C07304=1167.739,85.707,-51.427,-179.195,6.255,148.894
C07305=1167.744,85.458,-51.409,-179.197,6.253,148.894
C07306=1167.749,85.208,-51.392,-179.200,6.251,148.895
C07307=1167.754,84.959,-51.374,-179.203,6.251,148.895
C07308=1167.760,84.709,-51.357,-179.205,6.249,148.896
C07309=1167.764,84.460,-51.339,-179.208,6.248,148.896
C07310=1167.769,84.211,-51.321,-179.211,6.247,148.897
C07311=1167.774,83.961,-51.304,-179.213,6.246,148.897
C07312=1167.779,83.712,-51.286,-179.216,6.245,148.898
C07313=1167.784,83.463,-51.270,-179.218,6.244,148.898
C07314=1167.789,83.214,-51.252,-179.221,6.242,148.899
C07315=1167.794,82.964,-51.235,-179.224,6.241,148.899
C07316=1167.798,82.716,-51.217,-179.226,6.240,148.900
C07317=1167.803,82.466,-51.200,-179.230,6.239,148.900
C07318=1167.808,82.217,-51.182,-179.232,6.238,148.901
C07319=1167.813,81.967,-51.165,-179.234,6.236,148.901
C07320=1167.818,81.718,-51.147,-179.237,6.236,148.902
C07321=1167.823,81.468,-51.130,-179.240,6.234,148.902
C07322=1167.828,81.218,-51.113,-179.242,6.233,148.903
C07323=1167.832,80.969,-51.096,-179.245,6.232,148.903
C07324=1167.838,80.720,-51.079,-179.248,6.230,148.904
C07325=1167.843,80.452,-51.060,-179.250,6.229,148.904
C07326=1167.848,80.184,-51.041,-179.254,6.228,148.905
C07327=1167.854,79.915,-51.023,-179.256,6.226,148.905
C07328=1167.859,79.647,-51.004,-179.259,6.226,148.906
C07329=1167.863,79.398,-50.987,-179.262,6.224,148.907
C07330=1167.869,79.148,-50.969,-179.264,6.224,148.907
C07331=1167.874,78.898,-50.952,-179.267,6.222,148.908
C07332=1167.878,78.649,-50.935,-179.270,6.220,148.908
C07333=1167.884,78.400,-50.918,-179.272,6.220,148.909
C07334=1167.888,78.151,-50.901,-179.275,6.218,148.909
C07335=1167.893,77.901,-50.883,-179.278,6.218,148.910
C07336=1167.898,77.652,-50.866,-179.281,6.216,148.910
C07337=1167.903,77.402,-50.849,-179.283,6.215,148.911
C07338=1167.909,77.153,-50.832,-179.286,6.214,148.911
C07339=1167.913,76.904,-50.815,-179.288,6.213,148.912
C07340=1167.918,76.654,-50.798,-179.291,6.211,148.912
C07341=1167.923,76.405,-50.781,-179.293,6.211,148.913
C07342=1167.928,76.155,-50.764,-179.297,6.209,148.913
C07343=1167.932,75.906,-50.746,-179.299,6.208,148.914
C07344=1167.938,75.657,-50.730,-179.302,6.207,148.914
C07345=1167.942,75.408,-50.713,-179.304,6.206,148.915
C07346=1167.947,75.158,-50.696,-179.307,6.204,148.915
C07347=1167.952,74.908,-50.679,-179.310,6.204,148.916
C07348=1167.957,74.660,-50.661,-179.312,6.202,148.917
C07349=1167.962,74.410,-50.645,-179.315,6.202,148.917
C07350=1167.967,74.161,-50.627,-179.318,6.200,148.918
C07351=1167.972,73.911,-50.611,-179.320,6.199,148.918
C07352=1167.977,73.662,-50.594,-179.323,6.198,148.919
C07353=1167.982,73.413,-50.577,-179.325,6.197,148.919
C07354=1167.987,73.163,-50.560,-179.328,6.196,148.920
C07355=1167.991,72.914,-50.542,-179.330,6.195,148.920
C07356=1167.997,72.665,-50.526,-179.334,6.193,148.921
C07357=1168.002,72.415,-50.509,-179.336,6.192,148.921
C07358=1168.007,72.166,-50.492,-179.339,6.191,148.922
C07359=1168.011,71.916,-50.475,-179.341,6.190,148.922
C07360=1168.016,71.667,-50.459,-179.344,6.189,148.923
C07361=1168.022,71.418,-50.441,-179.347,6.188,148.923
C07362=1168.026,71.168,-50.425,-179.349,6.186,148.924
C07363=1168.031,70.918,-50.407,-179.352,6.186,148.925
C07364=1168.036,70.669,-50.391,-179.354,6.185,148.925
C07365=1168.041,70.420,-50.375,-179.357,6.184,148.926
C07366=1168.046,70.170,-50.357,-179.359,6.183,148.926
C07367=1168.051,69.921,-50.341,-179.362,6.181,148.927
C07368=1168.056,69.672,-50.324,-179.365,6.181,148.927
C07369=1168.061,69.422,-50.307,-179.368,6.179,148.928
C07370=1168.066,69.173,-50.291,-179.370,6.178,148.928
C07371=1168.071,68.924,-50.273,-179.373,6.177,148.929
C07372=1168.076,68.674,-50.257,-179.376,6.176,148.929
C07373=1168.081,68.425,-50.240,-179.378,6.175,148.930
C07374=1168.085,68.176,-50.224,-179.381,6.174,148.930
C07375=1168.090,67.926,-50.207,-179.384,6.172,148.931
C07376=1168.096,67.677,-50.190,-179.386,6.172,148.932
C07377=1168.100,67.427,-50.174,-179.388,6.171,148.932
C07378=1168.106,67.177,-50.157,-179.391,6.169,148.932
C07379=1168.111,66.929,-50.141,-179.394,6.169,148.933
C07380=1168.115,66.679,-50.124,-179.397,6.167,148.933
C07381=1168.120,66.429,-50.107,-179.399,6.167,148.934
C07382=1168.125,66.180,-50.090,-179.402,6.165,148.935
C07383=1168.130,65.931,-50.074,-179.405,6.164,148.935
C07384=1168.135,65.682,-50.058,-179.407,6.163,148.936
C07385=1168.140,65.432,-50.041,-179.410,6.162,148.936
C07386=1168.145,65.182,-50.024,-179.412,6.161,148.937
C07387=1168.150,64.934,-50.008,-179.415,6.160,148.937
C07388=1168.155,64.684,-49.991,-179.417,6.159,148.938
C07389=1168.160,64.435,-49.976,-179.421,6.158,148.939
C07390=1168.165,64.185,-49.958,-179.423,6.157,148.939
C07391=1168.170,63.935,-49.942,-179.426,6.156,148.940
C07392=1168.175,63.687,-49.926,-179.428,6.155,148.940
C07393=1168.179,63.436,-49.910,-179.431,6.153,148.940
C07394=1168.185,63.188,-49.893,-179.434,6.152,148.941
C07395=1168.190,62.938,-49.876,-179.436,6.152,148.942
C07396=1168.194,62.688,-49.859,-179.439,6.150,148.942
C07397=1168.200,62.439,-49.844,-179.441,6.149,148.943
C07398=1168.204,62.190,-49.827,-179.444,6.148,148.943
C07399=1168.209,61.941,-49.811,-179.446,6.147,148.944
C07400=1168.214,61.691,-49.795,-179.449,6.147,148.944
C07401=1168.220,61.442,-49.778,-179.452,6.145,148.945
C07402=1168.224,61.192,-49.761,-179.454,6.145,148.946
C07403=1168.230,60.943,-49.746,-179.457,6.143,148.946
C07404=1168.234,60.693,-49.729,-179.460,6.142,148.947
C07405=1168.239,60.444,-49.713,-179.462,6.141,148.947
C07406=1168.244,60.194,-49.697,-179.465,6.140,148.948
C07407=1168.249,59.946,-49.680,-179.467,6.139,148.948
C07408=1168.254,59.695,-49.664,-179.471,6.138,148.949
C07409=1168.259,59.447,-49.648,-179.473,6.137,148.949
C07410=1168.264,59.197,-49.631,-179.476,6.136,148.950
C07411=1168.270,58.947,-49.615,-179.478,6.135,148.950
C07412=1168.274,58.698,-49.599,-179.481,6.134,148.951
C07413=1168.279,58.449,-49.583,-179.483,6.133,148.951
C07414=1168.284,58.199,-49.566,-179.486,6.132,148.952
C07415=1168.289,57.950,-49.551,-179.488,6.131,148.953
C07416=1168.294,57.700,-49.534,-179.491,6.130,148.953
C07417=1168.299,57.451,-49.519,-179.494,6.129,148.954
C07418=1168.304,57.201,-49.502,-179.497,6.128,148.954
C07419=1168.309,56.952,-49.486,-179.499,6.127,148.955
C07420=1168.314,56.702,-49.470,-179.502,6.127,148.955
C07421=1168.319,56.453,-49.454,-179.504,6.125,148.956
C07422=1168.323,56.204,-49.437,-179.507,6.124,148.957
C07423=1168.329,55.954,-49.422,-179.510,6.123,148.957
C07424=1168.333,55.705,-49.405,-179.512,6.122,148.958
C07425=1168.339,55.455,-49.390,-179.515,6.121,148.958
C07426=1168.344,55.206,-49.373,-179.518,6.120,148.959
C07427=1168.349,54.956,-49.357,-179.520,6.119,148.959
C07428=1168.354,54.707,-49.342,-179.523,6.119,148.960
C07429=1168.359,54.438,-49.324,-179.525,6.117,148.960
C07430=1168.364,54.170,-49.307,-179.529,6.116,148.961
C07431=1168.370,53.901,-49.290,-179.531,6.115,148.962
C07432=1168.375,53.633,-49.273,-179.534,6.113,148.962
C07433=1168.380,53.383,-49.257,-179.537,6.113,148.963
C07434=1168.385,53.134,-49.240,-179.539,6.112,148.963
C07435=1168.390,52.885,-49.225,-179.542,6.111,148.964
C07436=1168.395,52.635,-49.209,-179.544,6.110,148.964
C07437=1168.400,52.386,-49.192,-179.547,6.109,148.965
C07438=1168.405,52.136,-49.176,-179.549,6.108,148.965
C07439=1168.410,51.887,-49.161,-179.552,6.107,148.966
C07440=1168.415,51.638,-49.145,-179.554,6.106,148.967
C07441=1168.420,51.388,-49.129,-179.557,6.105,148.967
C07442=1168.425,51.138,-49.114,-179.560,6.104,148.968
C07443=1168.430,50.889,-49.097,-179.562,6.104,148.968
C07444=1168.435,50.639,-49.081,-179.565,6.102,148.969
C07445=1168.440,50.390,-49.066,-179.568,6.102,148.969
C07446=1168.444,50.140,-49.050,-179.570,6.100,148.970
C07447=1168.449,49.891,-49.034,-179.573,6.099,148.971
C07448=1168.455,49.642,-49.019,-179.576,6.099,148.971
C07449=1168.460,49.392,-49.003,-179.578,6.097,148.972
C07450=1168.465,49.142,-48.987,-179.581,6.097,148.972
C07451=1168.470,48.893,-48.971,-179.583,6.096,148.973
C07452=1168.474,48.644,-48.955,-179.586,6.095,148.973
C07453=1168.479,48.395,-48.940,-179.589,6.094,148.974
C07454=1168.485,48.145,-48.924,-179.591,6.093,148.975
C07455=1168.490,47.895,-48.908,-179.594,6.091,148.975
C07456=1168.495,47.646,-48.893,-179.597,6.091,148.976
C07457=1168.500,47.397,-48.878,-179.599,6.090,148.976
C07458=1168.505,47.147,-48.862,-179.601,6.090,148.977
C07459=1168.510,46.898,-48.845,-179.604,6.088,148.977
C07460=1168.515,46.648,-48.830,-179.607,6.087,148.978
C07461=1168.520,46.399,-48.815,-179.609,6.087,148.978
C07462=1168.524,46.149,-48.799,-179.612,6.085,148.979
C07463=1168.530,45.900,-48.783,-179.614,6.084,148.979
C07464=1168.535,45.650,-48.768,-179.617,6.084,148.980
C07465=1168.540,45.401,-48.753,-179.620,6.082,148.981
C07466=1168.545,45.151,-48.737,-179.622,6.082,148.981
C07467=1168.550,44.902,-48.721,-179.624,6.081,148.982
C07468=1168.555,44.653,-48.706,-179.628,6.080,148.982
C07469=1168.559,44.402,-48.690,-179.630,6.079,148.983
C07470=1168.565,44.153,-48.675,-179.633,6.078,148.983
C07471=1168.570,43.904,-48.659,-179.636,6.077,148.984
C07472=1168.575,43.655,-48.644,-179.638,6.076,148.985
C07473=1168.580,43.405,-48.628,-179.641,6.076,148.985
C07474=1168.585,43.155,-48.612,-179.643,6.075,148.986
C07475=1168.590,42.906,-48.597,-179.646,6.073,148.986
C07476=1168.595,42.657,-48.582,-179.648,6.073,148.987
C07477=1168.600,42.407,-48.566,-179.651,6.072,148.987
C07478=1168.604,42.157,-48.551,-179.653,6.070,148.988
C07479=1168.610,41.908,-48.535,-179.656,6.070,148.989
C07480=1168.615,41.659,-48.520,-179.658,6.069,148.989
C07481=1168.620,41.409,-48.505,-179.661,6.069,148.990
C07482=1168.625,41.160,-48.489,-179.664,6.067,148.990
C07483=1168.629,40.910,-48.474,-179.666,6.066,148.991
C07484=1168.635,40.661,-48.458,-179.669,6.066,148.991
C07485=1168.640,40.411,-48.443,-179.672,6.064,148.992
C07486=1168.645,40.162,-48.428,-179.674,6.064,148.993
C07487=1168.650,39.912,-48.413,-179.676,6.063,148.993
C07488=1168.655,39.663,-48.398,-179.679,6.062,148.994
C07489=1168.660,39.413,-48.382,-179.682,6.061,148.994
C07490=1168.665,39.164,-48.367,-179.685,6.060,148.995
C07491=1168.670,38.915,-48.351,-179.687,6.059,148.995
C07492=1168.675,38.665,-48.336,-179.690,6.058,148.996
C07493=1168.680,38.416,-48.321,-179.693,6.058,148.997
C07494=1168.686,38.166,-48.306,-179.695,6.057,148.997
C07495=1168.690,37.916,-48.290,-179.697,6.056,148.998
C07496=1168.695,37.667,-48.275,-179.700,6.055,148.998
C07497=1168.700,37.417,-48.261,-179.703,6.054,148.999
C07498=1168.705,37.168,-48.245,-179.705,6.053,148.999
C07499=1168.710,36.919,-48.230,-179.708,6.053,149.000
C07500=1168.715,36.669,-48.214,-179.710,6.051,149.000
C07501=1168.720,36.420,-48.200,-179.713,6.051,149.001
C07502=1168.726,36.170,-48.185,-179.716,6.050,149.002
C07503=1168.730,35.920,-48.169,-179.718,6.049,149.002
C07504=1168.735,35.671,-48.154,-179.721,6.048,149.003
C07505=1168.740,35.421,-48.139,-179.723,6.047,149.003
C07506=1168.746,35.172,-48.124,-179.726,6.047,149.004
C07507=1168.750,34.923,-48.109,-179.728,6.046,149.004
C07508=1168.756,34.673,-48.094,-179.731,6.045,149.005
C07509=1168.761,34.424,-48.079,-179.733,6.044,149.006
C07510=1168.766,34.174,-48.063,-179.736,6.043,149.006
C07511=1168.771,33.925,-48.049,-179.739,6.043,149.007
C07512=1168.776,33.676,-48.034,-179.741,6.041,149.007
C07513=1168.781,33.426,-48.018,-179.744,6.041,149.008
C07514=1168.786,33.176,-48.004,-179.746,6.040,149.009
C07515=1168.791,32.927,-47.989,-179.749,6.039,149.009
C07516=1168.795,32.677,-47.973,-179.752,6.038,149.010
C07517=1168.800,32.427,-47.959,-179.754,6.037,149.010
C07518=1168.806,32.178,-47.943,-179.756,6.036,149.011
C07519=1168.811,31.928,-47.929,-179.759,6.036,149.011
C07520=1168.816,31.679,-47.913,-179.762,6.035,149.012
C07521=1168.821,31.429,-47.899,-179.764,6.034,149.013
C07522=1168.826,31.180,-47.884,-179.767,6.033,149.013
C07523=1168.831,30.931,-47.869,-179.769,6.032,149.014
C07524=1168.836,30.681,-47.854,-179.772,6.032,149.014
C07525=1168.841,30.432,-47.839,-179.775,6.030,149.015
C07526=1168.846,30.182,-47.824,-179.777,6.030,149.016
C07527=1168.851,29.933,-47.809,-179.780,6.029,149.016
C07528=1168.856,29.683,-47.795,-179.782,6.028,149.017
C07529=1168.861,29.434,-47.780,-179.785,6.028,149.017
C07530=1168.866,29.184,-47.765,-179.787,6.026,149.018
C07531=1168.871,28.935,-47.750,-179.790,6.026,149.018
C07532=1168.877,28.685,-47.735,-179.792,6.025,149.019
C07533=1168.882,28.416,-47.720,-179.795,6.024,149.020
C07534=1168.887,28.147,-47.704,-179.798,6.023,149.020
C07535=1168.893,27.878,-47.688,-179.801,6.023,149.021
C07536=1168.898,27.609,-47.672,-179.804,6.021,149.021
C07537=1168.903,27.360,-47.658,-179.806,6.020,149.022
C07538=1168.908,27.110,-47.642,-179.809,6.020,149.023
C07539=1168.913,26.861,-47.628,-179.811,6.019,149.023
C07540=1168.918,26.612,-47.613,-179.814,6.019,149.024
C07541=1168.923,26.363,-47.599,-179.816,6.017,149.024
C07542=1168.929,26.112,-47.584,-179.819,6.016,149.025
C07543=1168.934,25.863,-47.569,-179.822,6.016,149.026
C07544=1168.939,25.614,-47.555,-179.824,6.015,149.026
C07545=1168.944,25.364,-47.541,-179.827,6.015,149.027
C07546=1168.949,25.115,-47.525,-179.829,6.013,149.027
C07547=1168.954,24.865,-47.511,-179.832,6.013,149.028
C07548=1168.959,24.615,-47.496,-179.834,6.012,149.028
C07549=1168.964,24.366,-47.481,-179.837,6.011,149.029
C07550=1168.968,24.116,-47.467,-179.839,6.011,149.030
C07551=1168.974,23.866,-47.452,-179.842,6.010,149.030
C07552=1168.979,23.617,-47.437,-179.845,6.009,149.031
C07553=1168.984,23.368,-47.423,-179.847,6.008,149.031
C07554=1168.989,23.119,-47.409,-179.850,6.007,149.032
C07555=1168.994,22.869,-47.395,-179.852,6.006,149.032
C07556=1168.999,22.620,-47.380,-179.854,6.006,149.033
C07557=1169.005,22.370,-47.365,-179.857,6.005,149.034
C07558=1169.010,22.120,-47.351,-179.860,6.004,149.034
C07559=1169.015,21.870,-47.336,-179.862,6.003,149.035
C07560=1169.019,21.621,-47.321,-179.865,6.003,149.035
C07561=1169.024,21.371,-47.307,-179.867,6.002,149.036
C07562=1169.029,21.122,-47.293,-179.870,6.002,149.037
C07563=1169.035,20.873,-47.279,-179.872,6.001,149.037
C07564=1169.040,20.623,-47.265,-179.875,5.999,149.038
C07565=1169.045,20.374,-47.249,-179.877,5.999,149.038
C07566=1169.050,20.124,-47.235,-179.880,5.998,149.039
C07567=1169.055,19.874,-47.221,-179.883,5.998,149.040
C07568=1169.060,19.625,-47.206,-179.885,5.997,149.040
C07569=1169.065,19.375,-47.192,-179.888,5.996,149.041
C07570=1169.070,19.126,-47.178,-179.890,5.995,149.041
C07571=1169.075,18.876,-47.164,-179.893,5.994,149.042
C07572=1169.080,18.626,-47.150,-179.895,5.993,149.042
C07573=1169.085,18.377,-47.135,-179.898,5.993,149.043
C07574=1169.090,18.128,-47.120,-179.900,5.992,149.044
C07575=1169.095,17.879,-47.106,-179.903,5.992,149.044
C07576=1169.100,17.629,-47.092,-179.905,5.991,149.045
C07577=1169.105,17.379,-47.078,-179.908,5.989,149.045
C07578=1169.110,17.129,-47.063,-179.911,5.989,149.046
C07579=1169.115,16.880,-47.049,-179.913,5.989,149.047
C07580=1169.121,16.631,-47.035,-179.915,5.988,149.047
C07581=1169.126,16.381,-47.021,-179.918,5.987,149.048
C07582=1169.131,16.131,-47.007,-179.920,5.986,149.048
C07583=1169.136,15.882,-46.992,-179.923,5.986,149.049
C07584=1169.141,15.632,-46.978,-179.926,5.985,149.050
C07585=1169.146,15.383,-46.964,-179.928,5.984,149.050
C07586=1169.151,15.133,-46.950,-179.931,5.983,149.051
C07587=1169.156,14.883,-46.936,-179.933,5.982,149.051
C07588=1169.161,14.634,-46.921,-179.936,5.982,149.052
C07589=1169.167,14.385,-46.908,-179.938,5.982,149.053
C07590=1169.172,14.135,-46.893,-179.941,5.981,149.053
C07591=1169.177,13.885,-46.879,-179.943,5.980,149.054
C07592=1169.181,13.636,-46.865,-179.946,5.979,149.054
C07593=1169.187,13.387,-46.851,-179.949,5.978,149.055
C07594=1169.192,13.137,-46.837,-179.951,5.978,149.056
C07595=1169.197,12.887,-46.822,-179.954,5.977,149.056
C07596=1169.202,12.637,-46.808,-179.956,5.976,149.057
C07597=1169.208,12.388,-46.795,-179.958,5.975,149.057
C07598=1169.212,12.138,-46.781,-179.961,5.975,149.058
C07599=1169.217,11.889,-46.767,-179.964,5.975,149.059
C07600=1169.222,11.639,-46.753,-179.966,5.974,149.059
C07601=1169.227,11.390,-46.739,-179.969,5.972,149.060
C07602=1169.232,11.140,-46.724,-179.971,5.972,149.060
C07603=1169.237,10.891,-46.710,-179.974,5.971,149.061
C07604=1169.243,10.642,-46.696,-179.977,5.971,149.062
C07605=1169.248,10.391,-46.683,-179.979,5.970,149.062
C07606=1169.252,10.142,-46.669,-179.981,5.969,149.063
C07607=1169.258,9.893,-46.655,-179.984,5.969,149.063
C07608=1169.263,9.643,-46.641,-179.986,5.968,149.064
C07609=1169.268,9.393,-46.626,-179.989,5.968,149.065
C07610=1169.274,9.144,-46.613,-179.992,5.966,149.065
C07611=1169.279,8.894,-46.599,-179.994,5.965,149.066
C07612=1169.283,8.645,-46.585,-179.996,5.965,149.066
C07613=1169.288,8.396,-46.571,-179.999,5.964,149.067
C07614=1169.294,8.145,-46.558,179.998,5.964,149.068
C07615=1169.299,7.896,-46.544,179.996,5.963,149.068
C07616=1169.304,7.647,-46.530,179.993,5.962,149.069
C07617=1169.308,7.397,-46.516,179.991,5.962,149.069
C07618=1169.314,7.147,-46.502,179.989,5.961,149.070
C07619=1169.319,6.898,-46.488,179.986,5.961,149.071
C07620=1169.324,6.648,-46.474,179.984,5.960,149.071
C07621=1169.329,6.398,-46.461,179.981,5.959,149.072
C07622=1169.334,6.149,-46.447,179.978,5.958,149.072
C07623=1169.339,5.899,-46.433,179.976,5.957,149.073
C07624=1169.345,5.650,-46.420,179.973,5.957,149.074
C07625=1169.349,5.400,-46.406,179.971,5.956,149.074
C07626=1169.354,5.151,-46.392,179.968,5.955,149.075
C07627=1169.360,4.901,-46.379,179.966,5.955,149.075
C07628=1169.365,4.651,-46.364,179.963,5.954,149.076
C07629=1169.370,4.403,-46.351,179.961,5.954,149.076
C07630=1169.375,4.152,-46.338,179.959,5.953,149.077
C07631=1169.380,3.903,-46.323,179.956,5.952,149.078
C07632=1169.385,3.653,-46.311,179.954,5.952,149.078
C07633=1169.390,3.404,-46.296,179.951,5.951,149.079
C07634=1169.396,3.155,-46.282,179.949,5.951,149.079
C07635=1169.400,2.905,-46.270,179.946,5.950,149.080
C07636=1169.405,2.655,-46.255,179.944,5.949,149.081
C07637=1169.411,2.386,-46.241,179.940,5.948,149.081
C07638=1169.417,2.116,-46.226,179.938,5.948,149.082
C07639=1169.422,1.847,-46.211,179.936,5.947,149.082
C07640=1169.427,1.578,-46.197,179.933,5.946,149.083
C07641=1169.433,1.329,-46.183,179.930,5.946,149.084
C07642=1169.438,1.078,-46.169,179.928,5.945,149.084
C07643=1169.443,0.830,-46.156,179.925,5.945,149.085
C07644=1169.448,0.579,-46.143,179.922,5.943,149.086
C07645=1169.454,0.330,-46.129,179.920,5.943,149.086
C07646=1169.458,0.080,-46.116,179.917,5.942,149.087
C07647=1169.464,-0.169,-46.102,179.915,5.941,149.087
C07648=1169.468,-0.419,-46.089,179.913,5.941,149.088
C07649=1169.474,-0.668,-46.076,179.910,5.940,149.089
C07650=1169.479,-0.918,-46.061,179.908,5.939,149.089
C07651=1169.484,-1.168,-46.049,179.905,5.939,149.090
C07652=1169.489,-1.417,-46.034,179.903,5.938,149.090
C07653=1169.494,-1.667,-46.022,179.900,5.938,149.091
C07654=1169.499,-1.916,-46.008,179.898,5.937,149.092
C07655=1169.504,-2.166,-45.995,179.895,5.936,149.092
C07656=1169.510,-2.416,-45.981,179.893,5.936,149.093
C07657=1169.515,-2.665,-45.968,179.890,5.936,149.094
C07658=1169.520,-2.915,-45.955,179.888,5.935,149.094
C07659=1169.525,-3.164,-45.941,179.885,5.934,149.095
C07660=1169.530,-3.414,-45.928,179.883,5.933,149.095
C07661=1169.536,-3.664,-45.914,179.880,5.933,149.096
C07662=1169.540,-3.913,-45.901,179.878,5.933,149.096
C07663=1169.546,-4.163,-45.888,179.876,5.932,149.097
C07664=1169.550,-4.413,-45.875,179.873,5.931,149.098
C07665=1169.556,-4.662,-45.861,179.871,5.930,149.098
C07666=1169.560,-4.912,-45.848,179.868,5.930,149.099
C07667=1169.566,-5.161,-45.835,179.866,5.929,149.099
C07668=1169.571,-5.410,-45.821,179.863,5.929,149.100
C07669=1169.576,-5.660,-45.808,179.861,5.928,149.101
C07670=1169.581,-5.910,-45.795,179.858,5.928,149.101
C07671=1169.587,-6.160,-45.782,179.856,5.927,149.102
C07672=1169.591,-6.409,-45.768,179.853,5.926,149.102
C07673=1169.597,-6.659,-45.755,179.851,5.926,149.103
C07674=1169.602,-6.908,-45.742,179.848,5.925,149.104
C07675=1169.607,-7.158,-45.729,179.846,5.925,149.104
C07676=1169.612,-7.407,-45.715,179.844,5.924,149.105
C07677=1169.617,-7.657,-45.703,179.841,5.923,149.105
C07678=1169.622,-7.907,-45.689,179.839,5.923,149.106
C07679=1169.627,-8.156,-45.676,179.836,5.922,149.107
C07680=1169.633,-8.407,-45.663,179.833,5.922,149.107
C07681=1169.637,-8.655,-45.650,179.831,5.921,149.108
C07682=1169.643,-8.905,-45.637,179.829,5.920,149.108
C07683=1169.648,-9.155,-45.623,179.826,5.920,149.109
C07684=1169.653,-9.404,-45.611,179.824,5.919,149.110
C07685=1169.658,-9.654,-45.598,179.821,5.919,149.110
C07686=1169.663,-9.903,-45.584,179.819,5.918,149.111
C07687=1169.668,-10.153,-45.571,179.816,5.917,149.112
C07688=1169.673,-10.403,-45.558,179.814,5.917,149.112
C07689=1169.679,-10.652,-45.545,179.811,5.916,149.113
C07690=1169.684,-10.902,-45.533,179.809,5.916,149.113
C07691=1169.689,-11.152,-45.519,179.807,5.915,149.114
C07692=1169.694,-11.401,-45.506,179.804,5.914,149.115
C07693=1169.699,-11.651,-45.494,179.801,5.914,149.115
C07694=1169.704,-11.901,-45.480,179.799,5.913,149.116
C07695=1169.709,-12.150,-45.467,179.796,5.913,149.116
C07696=1169.714,-12.399,-45.454,179.794,5.912,149.117
C07697=1169.720,-12.649,-45.441,179.792,5.911,149.118
C07698=1169.725,-12.899,-45.428,179.789,5.911,149.118
C07699=1169.730,-13.148,-45.416,179.787,5.910,149.119
C07700=1169.734,-13.398,-45.403,179.784,5.910,149.119
C07701=1169.740,-13.648,-45.389,179.781,5.909,149.120
C07702=1169.745,-13.897,-45.377,179.779,5.908,149.121
C07703=1169.750,-14.147,-45.364,179.777,5.908,149.121
C07704=1169.756,-14.396,-45.351,179.774,5.907,149.122
C07705=1169.761,-14.646,-45.338,179.772,5.907,149.122
C07706=1169.765,-14.896,-45.325,179.769,5.906,149.123
C07707=1169.771,-15.145,-45.312,179.767,5.905,149.124
C07708=1169.776,-15.395,-45.299,179.764,5.905,149.124
C07709=1169.782,-15.644,-45.287,179.762,5.905,149.125
C07710=1169.786,-15.894,-45.274,179.759,5.904,149.125
C07711=1169.791,-16.143,-45.261,179.757,5.903,149.126
C07712=1169.797,-16.393,-45.248,179.755,5.902,149.127
C07713=1169.802,-16.643,-45.235,179.753,5.903,149.127
C07714=1169.807,-16.893,-45.223,179.750,5.902,149.128
C07715=1169.812,-17.142,-45.210,179.748,5.902,149.128
C07716=1169.817,-17.392,-45.198,179.745,5.901,149.129
C07717=1169.822,-17.642,-45.184,179.742,5.901,149.130
C07718=1169.828,-17.891,-45.172,179.740,5.900,149.130
C07719=1169.833,-18.141,-45.159,179.738,5.899,149.131
C07720=1169.838,-18.390,-45.146,179.735,5.899,149.131
C07721=1169.842,-18.640,-45.133,179.733,5.898,149.132
C07722=1169.848,-18.890,-45.120,179.730,5.898,149.133
C07723=1169.854,-19.140,-45.108,179.728,5.897,149.133
C07724=1169.859,-19.389,-45.096,179.725,5.896,149.134
C07725=1169.864,-19.638,-45.083,179.723,5.896,149.134
C07726=1169.868,-19.888,-45.070,179.720,5.895,149.135
C07727=1169.874,-20.137,-45.058,179.718,5.895,149.136
C07728=1169.879,-20.387,-45.044,179.716,5.894,149.136
C07729=1169.885,-20.637,-45.033,179.713,5.893,149.137
C07730=1169.889,-20.887,-45.020,179.711,5.894,149.138
C07731=1169.895,-21.136,-45.007,179.709,5.893,149.138
C07732=1169.900,-21.386,-44.994,179.706,5.893,149.139
C07733=1169.905,-21.636,-44.983,179.704,5.892,149.139
C07734=1169.910,-21.885,-44.970,179.701,5.891,149.140
C07735=1169.915,-22.135,-44.957,179.699,5.891,149.141
C07736=1169.921,-22.385,-44.944,179.696,5.890,149.141
C07737=1169.926,-22.635,-44.932,179.694,5.890,149.142
C07738=1169.931,-22.884,-44.919,179.691,5.889,149.142
C07739=1169.936,-23.133,-44.907,179.689,5.888,149.143
C07740=1169.941,-23.382,-44.894,179.686,5.888,149.144
C07741=1169.947,-23.653,-44.881,179.683,5.887,149.144
C07742=1169.952,-23.923,-44.867,179.681,5.887,149.145
C07743=1169.958,-24.193,-44.854,179.679,5.886,149.146
C07744=1169.963,-24.462,-44.841,179.676,5.886,149.146
C07745=1169.968,-24.712,-44.828,179.673,5.885,149.147
C07746=1169.974,-24.962,-44.816,179.671,5.885,149.147
C07747=1169.979,-25.211,-44.803,179.668,5.884,149.148
C07748=1169.984,-25.461,-44.790,179.666,5.883,149.149
C07749=1169.989,-25.711,-44.779,179.664,5.883,149.149
C07750=1169.994,-25.960,-44.766,179.662,5.883,149.150
C07751=1169.999,-26.209,-44.753,179.659,5.882,149.151
C07752=1170.005,-26.459,-44.742,179.657,5.882,149.151
C07753=1170.010,-26.709,-44.729,179.654,5.882,149.152
C07754=1170.015,-26.958,-44.716,179.652,5.881,149.152
C07755=1170.020,-27.208,-44.704,179.649,5.880,149.153
C07756=1170.025,-27.458,-44.691,179.647,5.879,149.154
C07757=1170.030,-27.708,-44.680,179.644,5.879,149.154
C07758=1170.035,-27.957,-44.667,179.642,5.879,149.155
C07759=1170.041,-28.207,-44.655,179.640,5.878,149.155
C07760=1170.046,-28.456,-44.642,179.637,5.878,149.156
C07761=1170.051,-28.706,-44.630,179.635,5.877,149.157
C07762=1170.056,-28.956,-44.618,179.633,5.877,149.157
C07763=1170.062,-29.205,-44.605,179.630,5.876,149.158
C07764=1170.067,-29.455,-44.594,179.628,5.876,149.158
C07765=1170.072,-29.704,-44.581,179.625,5.875,149.159
C07766=1170.078,-29.954,-44.569,179.623,5.874,149.160
C07767=1170.082,-30.204,-44.556,179.620,5.874,149.160
C07768=1170.088,-30.454,-44.544,179.618,5.874,149.161
C07769=1170.092,-30.703,-44.532,179.616,5.873,149.161
C07770=1170.097,-30.953,-44.520,179.613,5.873,149.162
C07771=1170.102,-31.202,-44.508,179.611,5.873,149.163
C07772=1170.108,-31.452,-44.496,179.609,5.872,149.163
C07773=1170.113,-31.702,-44.483,179.606,5.871,149.164
C07774=1170.118,-31.952,-44.471,179.604,5.871,149.165
C07775=1170.124,-32.202,-44.459,179.601,5.870,149.165
C07776=1170.129,-32.451,-44.447,179.598,5.870,149.166
C07777=1170.134,-32.701,-44.436,179.597,5.870,149.166
C07778=1170.139,-32.950,-44.423,179.594,5.869,149.167
C07779=1170.144,-33.200,-44.411,179.592,5.868,149.168
C07780=1170.150,-33.450,-44.399,179.589,5.868,149.168
C07781=1170.155,-33.699,-44.387,179.587,5.868,149.169
C07782=1170.160,-33.949,-44.375,179.584,5.867,149.169
C07783=1170.165,-34.198,-44.362,179.582,5.866,149.170
C07784=1170.170,-34.448,-44.351,179.580,5.866,149.171
C07785=1170.176,-34.698,-44.339,179.578,5.866,149.171
C07786=1170.181,-34.947,-44.326,179.575,5.865,149.172
C07787=1170.186,-35.197,-44.314,179.573,5.865,149.172
C07788=1170.191,-35.447,-44.303,179.570,5.864,149.173
C07789=1170.196,-35.696,-44.291,179.567,5.864,149.174
C07790=1170.201,-35.946,-44.279,179.565,5.863,149.174
C07791=1170.207,-36.196,-44.267,179.563,5.863,149.175
C07792=1170.212,-36.445,-44.254,179.561,5.863,149.176
C07793=1170.217,-36.695,-44.242,179.558,5.862,149.176
C07794=1170.222,-36.945,-44.231,179.556,5.862,149.177
C07795=1170.227,-37.194,-44.218,179.553,5.861,149.177
C07796=1170.233,-37.444,-44.206,179.551,5.860,149.178
C07797=1170.238,-37.694,-44.195,179.549,5.860,149.179
C07798=1170.243,-37.944,-44.183,179.547,5.860,149.179
C07799=1170.248,-38.193,-44.171,179.544,5.860,149.180
C07800=1170.253,-38.443,-44.159,179.542,5.859,149.180
C07801=1170.259,-38.693,-44.147,179.539,5.858,149.181
C07802=1170.264,-38.942,-44.136,179.537,5.858,149.182
C07803=1170.269,-39.191,-44.123,179.534,5.857,149.182
C07804=1170.274,-39.441,-44.112,179.532,5.857,149.183
C07805=1170.280,-39.691,-44.100,179.530,5.857,149.183
C07806=1170.285,-39.941,-44.088,179.527,5.856,149.184
C07807=1170.290,-40.190,-44.076,179.525,5.855,149.185
C07808=1170.295,-40.440,-44.064,179.522,5.855,149.185
C07809=1170.300,-40.689,-44.053,179.520,5.855,149.186
C07810=1170.305,-40.939,-44.041,179.518,5.855,149.187
C07811=1170.311,-41.189,-44.029,179.515,5.854,149.187
C07812=1170.315,-41.439,-44.018,179.513,5.853,149.188
C07813=1170.321,-41.688,-44.006,179.511,5.853,149.188
C07814=1170.327,-41.938,-43.994,179.508,5.852,149.189
C07815=1170.331,-42.187,-43.982,179.506,5.852,149.190
C07816=1170.337,-42.437,-43.970,179.504,5.852,149.190
C07817=1170.342,-42.687,-43.958,179.502,5.851,149.191
C07818=1170.347,-42.937,-43.947,179.499,5.851,149.191
C07819=1170.352,-43.187,-43.935,179.496,5.850,149.192
C07820=1170.358,-43.436,-43.923,179.494,5.850,149.193
C07821=1170.362,-43.686,-43.912,179.492,5.850,149.193
C07822=1170.368,-43.935,-43.900,179.490,5.849,149.194
C07823=1170.373,-44.185,-43.889,179.487,5.849,149.195
C07824=1170.378,-44.435,-43.877,179.484,5.848,149.195
C07825=1170.384,-44.684,-43.865,179.482,5.847,149.196
C07826=1170.388,-44.934,-43.853,179.480,5.847,149.196
C07827=1170.394,-45.184,-43.842,179.478,5.847,149.197
C07828=1170.398,-45.433,-43.830,179.475,5.847,149.198
C07829=1170.404,-45.683,-43.819,179.473,5.846,149.198
C07830=1170.409,-45.932,-43.807,179.470,5.845,149.199
C07831=1170.415,-46.182,-43.796,179.468,5.845,149.199
C07832=1170.420,-46.432,-43.784,179.466,5.845,149.200
C07833=1170.425,-46.682,-43.772,179.464,5.845,149.201
C07834=1170.430,-46.932,-43.760,179.461,5.844,149.201
C07835=1170.435,-47.181,-43.750,179.459,5.843,149.202
C07836=1170.441,-47.431,-43.738,179.456,5.843,149.203
C07837=1170.446,-47.680,-43.726,179.454,5.843,149.203
C07838=1170.451,-47.930,-43.714,179.452,5.842,149.204
C07839=1170.456,-48.180,-43.703,179.449,5.842,149.204
C07840=1170.462,-48.430,-43.692,179.447,5.841,149.205
C07841=1170.467,-48.679,-43.681,179.444,5.841,149.206
C07842=1170.472,-48.929,-43.669,179.443,5.841,149.206
C07843=1170.478,-49.179,-43.657,179.440,5.840,149.207
C07844=1170.483,-49.428,-43.646,179.438,5.840,149.207
C07845=1170.488,-49.698,-43.633,179.435,5.839,149.208
C07846=1170.494,-49.969,-43.621,179.432,5.839,149.209
C07847=1170.500,-50.240,-43.609,179.430,5.838,149.209
C07848=1170.505,-50.510,-43.596,179.427,5.838,149.210
C07849=1170.510,-50.760,-43.585,179.426,5.838,149.211
C07850=1170.515,-51.010,-43.573,179.423,5.838,149.211
C07851=1170.521,-51.259,-43.563,179.421,5.837,149.212
C07852=1170.526,-51.509,-43.551,179.418,5.836,149.212
C07853=1170.531,-51.759,-43.540,179.415,5.836,149.213
C07854=1170.536,-52.008,-43.529,179.414,5.836,149.214
C07855=1170.542,-52.258,-43.517,179.411,5.835,149.214
C07856=1170.547,-52.507,-43.506,179.409,5.835,149.215
C07857=1170.552,-52.758,-43.495,179.406,5.834,149.215
C07858=1170.558,-53.007,-43.484,179.404,5.835,149.216
C07859=1170.563,-53.257,-43.472,179.402,5.834,149.217
C07860=1170.568,-53.506,-43.460,179.399,5.833,149.217
C07861=1170.572,-53.756,-43.449,179.397,5.833,149.218
C07862=1170.579,-54.006,-43.438,179.394,5.832,149.219
C07863=1170.583,-54.255,-43.427,179.393,5.832,149.219
C07864=1170.589,-54.505,-43.415,179.390,5.832,149.220
C07865=1170.594,-54.755,-43.404,179.388,5.831,149.220
C07866=1170.599,-55.004,-43.394,179.385,5.831,149.221
C07867=1170.605,-55.254,-43.382,179.383,5.831,149.222
C07868=1170.609,-55.504,-43.370,179.381,5.830,149.222
C07869=1170.615,-55.753,-43.360,179.378,5.830,149.223
C07870=1170.620,-56.003,-43.348,179.376,5.829,149.223
C07871=1170.625,-56.253,-43.337,179.374,5.829,149.224
C07872=1170.630,-56.502,-43.326,179.371,5.829,149.225
C07873=1170.636,-56.752,-43.314,179.369,5.828,149.225
C07874=1170.641,-57.002,-43.304,179.367,5.828,149.226
C07875=1170.645,-57.252,-43.292,179.365,5.828,149.226
C07876=1170.651,-57.501,-43.281,179.362,5.827,149.227
C07877=1170.656,-57.751,-43.270,179.360,5.827,149.228
C07878=1170.661,-58.001,-43.259,179.358,5.826,149.228
C07879=1170.667,-58.250,-43.248,179.355,5.826,149.229
C07880=1170.672,-58.500,-43.237,179.353,5.826,149.229
C07881=1170.677,-58.750,-43.226,179.351,5.825,149.230
C07882=1170.682,-58.999,-43.215,179.348,5.824,149.231
C07883=1170.688,-59.249,-43.204,179.346,5.825,149.231
C07884=1170.693,-59.499,-43.192,179.344,5.824,149.232
C07885=1170.698,-59.749,-43.182,179.341,5.824,149.232
C07886=1170.704,-59.999,-43.170,179.339,5.823,149.233
C07887=1170.709,-60.248,-43.159,179.337,5.823,149.234
C07888=1170.714,-60.498,-43.149,179.335,5.823,149.234
C07889=1170.719,-60.747,-43.137,179.332,5.822,149.235
C07890=1170.725,-60.997,-43.127,179.330,5.822,149.236
C07891=1170.730,-61.247,-43.115,179.328,5.822,149.236
C07892=1170.735,-61.497,-43.105,179.325,5.821,149.237
C07893=1170.740,-61.746,-43.094,179.323,5.821,149.237
C07894=1170.745,-61.996,-43.082,179.321,5.821,149.238
C07895=1170.751,-62.246,-43.072,179.319,5.820,149.239
C07896=1170.756,-62.495,-43.060,179.316,5.820,149.239
C07897=1170.761,-62.745,-43.050,179.314,5.819,149.240
C07898=1170.766,-62.994,-43.039,179.312,5.820,149.240
C07899=1170.772,-63.245,-43.028,179.309,5.819,149.241
C07900=1170.777,-63.494,-43.017,179.307,5.818,149.242
C07901=1170.782,-63.744,-43.006,179.305,5.818,149.242
C07902=1170.787,-63.994,-42.995,179.302,5.818,149.243
C07903=1170.792,-64.243,-42.985,179.300,5.817,149.243
C07904=1170.798,-64.493,-42.973,179.298,5.817,149.244
C07905=1170.803,-64.743,-42.963,179.296,5.817,149.245
C07906=1170.808,-64.992,-42.951,179.293,5.816,149.245
C07907=1170.814,-65.242,-42.941,179.291,5.816,149.246
C07908=1170.819,-65.492,-42.931,179.288,5.815,149.246
C07909=1170.824,-65.741,-42.920,179.286,5.815,149.247
C07910=1170.830,-65.992,-42.908,179.284,5.815,149.248
C07911=1170.834,-66.241,-42.897,179.282,5.814,149.248
C07912=1170.840,-66.491,-42.887,179.280,5.814,149.249
C07913=1170.845,-66.740,-42.876,179.277,5.814,149.249
C07914=1170.850,-66.990,-42.865,179.275,5.813,149.250
C07915=1170.855,-67.240,-42.855,179.272,5.813,149.251
C07916=1170.860,-67.489,-42.844,179.270,5.813,149.251
C07917=1170.865,-67.739,-42.833,179.268,5.812,149.252
C07918=1170.872,-67.989,-42.823,179.265,5.812,149.253
C07919=1170.876,-68.239,-42.811,179.264,5.812,149.253
C07920=1170.882,-68.488,-42.801,179.261,5.811,149.254
C07921=1170.887,-68.739,-42.791,179.259,5.811,149.254
C07922=1170.892,-68.988,-42.780,179.256,5.810,149.255
C07923=1170.897,-69.238,-42.769,179.255,5.810,149.255
C07924=1170.903,-69.487,-42.759,179.252,5.810,149.256
C07925=1170.908,-69.737,-42.748,179.250,5.809,149.257
C07926=1170.913,-69.986,-42.737,179.248,5.809,149.257
C07927=1170.918,-70.237,-42.727,179.245,5.809,149.258
C07928=1170.924,-70.486,-42.716,179.243,5.808,149.259
C07929=1170.929,-70.736,-42.705,179.241,5.809,149.259
C07930=1170.934,-70.985,-42.695,179.239,5.808,149.260
C07931=1170.940,-71.235,-42.683,179.236,5.807,149.260
C07932=1170.945,-71.485,-42.673,179.234,5.807,149.261
C07933=1170.950,-71.735,-42.662,179.232,5.807,149.262
C07934=1170.956,-71.985,-42.652,179.230,5.806,149.262
C07935=1170.960,-72.234,-42.641,179.227,5.806,149.263
C07936=1170.966,-72.484,-42.631,179.225,5.806,149.263
C07937=1170.972,-72.733,-42.620,179.223,5.805,149.264
C07938=1170.977,-72.984,-42.610,179.220,5.805,149.265
C07939=1170.982,-73.233,-42.599,179.218,5.805,149.265
C07940=1170.987,-73.483,-42.588,179.216,5.805,149.266
C07941=1170.993,-73.732,-42.578,179.214,5.804,149.266
C07942=1170.998,-73.983,-42.568,179.211,5.804,149.267
C07943=1171.003,-74.232,-42.557,179.209,5.804,149.268
C07944=1171.008,-74.482,-42.546,179.207,5.803,149.268
C07945=1171.013,-74.731,-42.536,179.205,5.803,149.269
C07946=1171.019,-74.981,-42.526,179.202,5.803,149.269
C07947=1171.024,-75.231,-42.515,179.200,5.802,149.270
C07948=1171.030,-75.481,-42.505,179.198,5.802,149.271
C07949=1171.035,-75.752,-42.494,179.195,5.802,149.271
C07950=1171.040,-76.023,-42.482,179.193,5.801,149.272
C07951=1171.046,-76.294,-42.471,179.191,5.801,149.273
C07952=1171.052,-76.565,-42.460,179.188,5.800,149.273
C07953=1171.058,-76.815,-42.449,179.186,5.800,149.274
C07954=1171.063,-77.065,-42.439,179.184,5.800,149.274
C07955=1171.068,-77.314,-42.429,179.181,5.799,149.275
C07956=1171.074,-77.564,-42.418,179.179,5.800,149.276
C07957=1171.079,-77.814,-42.407,179.177,5.799,149.276
C07958=1171.083,-78.063,-42.398,179.174,5.798,149.277
C07959=1171.088,-78.313,-42.387,179.172,5.799,149.277
C07960=1171.094,-78.563,-42.377,179.170,5.798,149.278
C07961=1171.100,-78.812,-42.367,179.168,5.798,149.279
C07962=1171.105,-79.062,-42.356,179.166,5.798,149.279
C07963=1171.110,-79.312,-42.346,179.163,5.797,149.280
C07964=1171.116,-79.562,-42.336,179.161,5.796,149.280
C07965=1171.121,-79.812,-42.325,179.159,5.797,149.281
C07966=1171.126,-80.061,-42.315,179.157,5.796,149.282
C07967=1171.131,-80.311,-42.305,179.154,5.796,149.282
C07968=1171.136,-80.561,-42.295,179.153,5.796,149.283
C07969=1171.142,-80.810,-42.284,179.150,5.795,149.283
C07970=1171.147,-81.060,-42.274,179.148,5.795,149.284
C07971=1171.152,-81.310,-42.264,179.146,5.795,149.285
C07972=1171.158,-81.560,-42.253,179.143,5.794,149.285
C07973=1171.163,-81.809,-42.244,179.141,5.794,149.286
C07974=1171.168,-82.059,-42.233,179.139,5.794,149.286
C07975=1171.174,-82.309,-42.223,179.136,5.793,149.287
C07976=1171.179,-82.558,-42.213,179.135,5.793,149.288
C07977=1171.184,-82.808,-42.202,179.132,5.793,149.288
C07978=1171.189,-83.058,-42.193,179.130,5.792,149.289
C07979=1171.195,-83.307,-42.182,179.128,5.793,149.289
C07980=1171.200,-83.557,-42.172,179.126,5.792,149.290
C07981=1171.205,-83.807,-42.162,179.123,5.791,149.291
C07982=1171.211,-84.057,-42.151,179.121,5.791,149.291
C07983=1171.215,-84.307,-42.141,179.119,5.791,149.292
C07984=1171.221,-84.557,-42.132,179.117,5.791,149.292
C07985=1171.227,-84.806,-42.122,179.115,5.791,149.293
C07986=1171.232,-85.056,-42.111,179.112,5.790,149.293
C07987=1171.236,-85.306,-42.101,179.110,5.790,149.294
C07988=1171.242,-85.555,-42.091,179.108,5.789,149.295
C07989=1171.248,-85.805,-42.081,179.105,5.789,149.295
C07990=1171.253,-86.055,-42.070,179.104,5.789,149.296
C07991=1171.257,-86.304,-42.061,179.101,5.789,149.297
C07992=1171.263,-86.554,-42.051,179.099,5.788,149.297
C07993=1171.268,-86.805,-42.041,179.097,5.788,149.298
C07994=1171.274,-87.054,-42.031,179.095,5.787,149.298
C07995=1171.279,-87.303,-42.021,179.093,5.788,149.299
C07996=1171.284,-87.553,-42.011,179.090,5.787,149.299
C07997=1171.289,-87.803,-42.000,179.088,5.787,149.300
C07998=1171.295,-88.053,-41.991,179.086,5.787,149.301
C07999=1171.300,-88.303,-41.981,179.083,5.786,149.301
C08000=1171.306,-88.552,-41.971,179.081,5.786,149.302
C08001=1171.310,-88.802,-41.961,179.079,5.786,149.303
C08002=1171.316,-89.052,-41.951,179.077,5.785,149.303
C08003=1171.322,-89.302,-41.941,179.075,5.786,149.304
C08004=1171.326,-89.551,-41.932,179.073,5.785,149.304
C08005=1171.332,-89.801,-41.921,179.070,5.784,149.305
C08006=1171.337,-90.051,-41.911,179.068,5.784,149.305
C08007=1171.342,-90.301,-41.902,179.066,5.784,149.306
C08008=1171.348,-90.550,-41.892,179.064,5.784,149.307
C08009=1171.353,-90.800,-41.882,179.062,5.784,149.307
C08010=1171.358,-91.050,-41.872,179.059,5.783,149.308
C08011=1171.364,-91.300,-41.862,179.057,5.783,149.308
C08012=1171.369,-91.549,-41.852,179.055,5.782,149.309
C08013=1171.374,-91.799,-41.842,179.053,5.783,149.310
C08014=1171.380,-92.049,-41.833,179.051,5.782,149.310
C08015=1171.384,-92.299,-41.823,179.049,5.781,149.311
C08016=1171.390,-92.548,-41.813,179.047,5.782,149.311
C08017=1171.396,-92.798,-41.803,179.044,5.781,149.312
C08018=1171.401,-93.048,-41.793,179.042,5.781,149.313
C08019=1171.406,-93.297,-41.783,179.040,5.781,149.313
C08020=1171.412,-93.547,-41.774,179.037,5.780,149.314
C08021=1171.416,-93.797,-41.764,179.036,5.780,149.314
C08022=1171.422,-94.047,-41.754,179.033,5.780,149.315
C08023=1171.427,-94.297,-41.745,179.031,5.779,149.315
C08024=1171.433,-94.546,-41.734,179.029,5.779,149.316
C08025=1171.438,-94.795,-41.725,179.027,5.779,149.317
C08026=1171.443,-95.046,-41.715,179.025,5.779,149.317
C08027=1171.448,-95.296,-41.705,179.022,5.778,149.318
C08028=1171.454,-95.546,-41.696,179.020,5.779,149.319
C08029=1171.459,-95.795,-41.686,179.018,5.778,149.319
C08030=1171.464,-96.045,-41.676,179.015,5.778,149.320
C08031=1171.470,-96.295,-41.667,179.014,5.778,149.320
C08032=1171.475,-96.544,-41.657,179.012,5.777,149.321
C08033=1171.481,-96.794,-41.647,179.010,5.777,149.321
C08034=1171.485,-97.044,-41.637,179.007,5.776,149.322
C08035=1171.491,-97.294,-41.627,179.005,5.776,149.323
C08036=1171.496,-97.543,-41.618,179.003,5.776,149.323
C08037=1171.501,-97.793,-41.608,179.000,5.776,149.324
C08038=1171.506,-98.043,-41.599,178.999,5.776,149.324
C08039=1171.512,-98.292,-41.589,178.996,5.775,149.325
C08040=1171.518,-98.542,-41.580,178.994,5.775,149.325
C08041=1171.523,-98.792,-41.570,178.992,5.775,149.326
C08042=1171.529,-99.042,-41.560,178.990,5.774,149.327
C08043=1171.534,-99.291,-41.551,178.988,5.774,149.327
C08044=1171.538,-99.542,-41.542,178.985,5.774,149.328
C08045=1171.544,-99.791,-41.531,178.984,5.774,149.328
C08046=1171.549,-100.041,-41.522,178.981,5.773,149.329
C08047=1171.555,-100.291,-41.512,178.979,5.773,149.330
C08048=1171.560,-100.540,-41.503,178.977,5.773,149.330
C08049=1171.565,-100.790,-41.493,178.975,5.772,149.331
C08050=1171.570,-101.040,-41.484,178.973,5.773,149.331
C08051=1171.576,-101.289,-41.474,178.970,5.772,149.332
C08052=1171.581,-101.539,-41.465,178.969,5.772,149.332
C08053=1171.587,-101.811,-41.455,178.966,5.772,149.333
C08054=1171.593,-102.083,-41.444,178.963,5.771,149.334
C08055=1171.598,-102.355,-41.434,178.961,5.770,149.334
C08056=1171.605,-102.627,-41.424,178.959,5.771,149.335
C08057=1171.609,-102.876,-41.414,178.957,5.770,149.336
C08058=1171.615,-103.127,-41.405,178.955,5.770,149.336
C08059=1171.620,-103.377,-41.396,178.953,5.770,149.337
C08060=1171.625,-103.626,-41.385,178.950,5.769,149.337
C08061=1171.631,-103.876,-41.377,178.948,5.769,149.338
C08062=1171.636,-104.125,-41.367,178.946,5.769,149.339
C08063=1171.641,-104.375,-41.357,178.944,5.769,149.339
C08064=1171.647,-104.625,-41.349,178.942,5.768,149.340
C08065=1171.651,-104.874,-41.339,178.940,5.769,149.340
C08066=1171.657,-105.125,-41.329,178.938,5.768,149.341
C08067=1171.663,-105.374,-41.320,178.936,5.768,149.342
C08068=1171.668,-105.624,-41.310,178.933,5.767,149.342
C08069=1171.673,-105.874,-41.301,178.931,5.767,149.343
C08070=1171.678,-106.124,-41.292,178.929,5.767,149.343
C08071=1171.684,-106.373,-41.282,178.927,5.766,149.344
C08072=1171.689,-106.623,-41.273,178.925,5.767,149.344
C08073=1171.694,-106.873,-41.264,178.923,5.766,149.345
C08074=1171.700,-107.122,-41.254,178.921,5.766,149.346
C08075=1171.705,-107.372,-41.245,178.918,5.766,149.346
C08076=1171.710,-107.622,-41.236,178.917,5.766,149.347
C08077=1171.716,-107.872,-41.227,178.914,5.765,149.347
C08078=1171.721,-108.122,-41.217,178.913,5.765,149.348
C08079=1171.726,-108.371,-41.208,178.910,5.765,149.349
C08080=1171.732,-108.622,-41.199,178.908,5.764,149.349
C08081=1171.737,-108.871,-41.190,178.906,5.765,149.350
C08082=1171.742,-109.121,-41.180,178.903,5.764,149.350
C08083=1171.747,-109.370,-41.172,178.902,5.764,149.351
C08084=1171.753,-109.621,-41.162,178.899,5.763,149.351
C08085=1171.758,-109.870,-41.153,178.898,5.763,149.352
C08086=1171.763,-110.120,-41.144,178.895,5.763,149.353
C08087=1171.769,-110.370,-41.134,178.893,5.763,149.353
C08088=1171.774,-110.620,-41.125,178.891,5.762,149.354
C08089=1171.780,-110.870,-41.116,178.889,5.763,149.354
C08090=1171.785,-111.119,-41.108,178.887,5.762,149.355
C08091=1171.791,-111.368,-41.098,178.884,5.762,149.355
C08092=1171.796,-111.618,-41.089,178.882,5.762,149.356
C08093=1171.801,-111.868,-41.080,178.880,5.761,149.356
C08094=1171.806,-112.118,-41.071,178.878,5.761,149.357
C08095=1171.812,-112.368,-41.061,178.876,5.760,149.358
C08096=1171.817,-112.618,-41.052,178.874,5.761,149.358
C08097=1171.822,-112.867,-41.043,178.872,5.760,149.359
C08098=1171.827,-113.117,-41.034,178.870,5.760,149.359
C08099=1171.833,-113.367,-41.025,178.867,5.760,149.360
C08100=1171.839,-113.617,-41.016,178.866,5.760,149.361
C08101=1171.844,-113.867,-41.007,178.864,5.759,149.361
C08102=1171.849,-114.117,-40.998,178.862,5.759,149.362
C08103=1171.855,-114.366,-40.989,178.859,5.759,149.362
C08104=1171.860,-114.616,-40.980,178.857,5.759,149.363
C08105=1171.865,-114.865,-40.970,178.855,5.758,149.363
C08106=1171.871,-115.115,-40.961,178.854,5.758,149.364
C08107=1171.876,-115.365,-40.952,178.851,5.758,149.365
C08108=1171.881,-115.615,-40.943,178.849,5.758,149.365
C08109=1171.886,-115.865,-40.935,178.847,5.757,149.366
C08110=1171.892,-116.115,-40.925,178.844,5.757,149.366
C08111=1171.897,-116.365,-40.916,178.843,5.757,149.367
C08112=1171.903,-116.614,-40.908,178.840,5.757,149.368
C08113=1171.908,-116.864,-40.899,178.839,5.757,149.368
C08114=1171.913,-117.113,-40.890,178.836,5.756,149.368
C08115=1171.918,-117.363,-40.881,178.834,5.756,149.369
C08116=1171.924,-117.613,-40.872,178.832,5.755,149.370
C08117=1171.929,-117.863,-40.863,178.830,5.755,149.370
C08118=1171.935,-118.113,-40.854,178.828,5.755,149.371
C08119=1171.940,-118.362,-40.845,178.826,5.755,149.371
C08120=1171.946,-118.612,-40.836,178.824,5.754,149.372
C08121=1171.951,-118.862,-40.827,178.822,5.755,149.373
C08122=1171.956,-119.112,-40.818,178.820,5.754,149.373
C08123=1171.961,-119.362,-40.809,178.818,5.754,149.374
C08124=1171.966,-119.612,-40.801,178.815,5.754,149.374
C08125=1171.971,-119.861,-40.792,178.814,5.754,149.375
C08126=1171.978,-120.111,-40.783,178.811,5.753,149.375
C08127=1171.983,-120.361,-40.774,178.810,5.753,149.376
C08128=1171.988,-120.611,-40.765,178.807,5.753,149.376
C08129=1171.993,-120.860,-40.756,178.805,5.753,149.377
C08130=1171.999,-121.110,-40.747,178.803,5.752,149.378
C08131=1172.004,-121.359,-40.738,178.801,5.752,149.378
C08132=1172.010,-121.609,-40.730,178.799,5.752,149.379
C08133=1172.015,-121.859,-40.721,178.797,5.752,149.379
C08134=1172.020,-122.109,-40.712,178.795,5.751,149.380
C08135=1172.025,-122.359,-40.704,178.793,5.752,149.381
C08136=1172.030,-122.609,-40.695,178.791,5.751,149.381
C08137=1172.036,-122.858,-40.686,178.789,5.751,149.382
C08138=1172.041,-123.108,-40.677,178.786,5.750,149.382
C08139=1172.047,-123.358,-40.668,178.785,5.750,149.383
C08140=1172.052,-123.608,-40.659,178.783,5.750,149.383
C08141=1172.058,-123.857,-40.651,178.781,5.750,149.384
C08142=1172.063,-124.107,-40.642,178.778,5.749,149.384
C08143=1172.068,-124.357,-40.634,178.777,5.749,149.385
C08144=1172.073,-124.607,-40.625,178.774,5.749,149.386
C08145=1172.078,-124.857,-40.616,178.772,5.749,149.386
C08146=1172.084,-125.106,-40.608,178.770,5.748,149.387
C08147=1172.089,-125.356,-40.599,178.768,5.749,149.387
C08148=1172.095,-125.606,-40.590,178.766,5.748,149.388
C08149=1172.100,-125.857,-40.582,178.764,5.748,149.388
C08150=1172.106,-126.106,-40.573,178.762,5.748,149.389
C08151=1172.111,-126.356,-40.564,178.760,5.748,149.389
C08152=1172.116,-126.605,-40.555,178.758,5.747,149.390
C08153=1172.121,-126.855,-40.546,178.756,5.747,149.391
C08154=1172.127,-127.105,-40.538,178.754,5.747,149.391
C08155=1172.133,-127.355,-40.530,178.752,5.747,149.392
C08156=1172.138,-127.605,-40.521,178.750,5.747,149.392
C08157=1171.717,-127.616,-40.562,178.746,5.750,149.394
C08158=1171.711,-127.365,-40.570,178.748,5.750,149.394
C08159=1171.706,-127.116,-40.579,178.750,5.751,149.393
C08160=1171.701,-126.866,-40.587,178.752,5.751,149.393
C08161=1171.695,-126.617,-40.596,178.755,5.751,149.392
C08162=1171.690,-126.366,-40.605,178.756,5.751,149.391
C08163=1171.684,-126.117,-40.613,178.758,5.752,149.391
C08164=1171.679,-125.867,-40.622,178.761,5.751,149.390
C08165=1171.674,-125.617,-40.631,178.763,5.752,149.390
C08166=1171.669,-125.367,-40.640,178.764,5.752,149.389
C08167=1171.663,-125.118,-40.648,178.767,5.752,149.388
C08168=1171.657,-124.868,-40.656,178.769,5.752,149.388
C08169=1171.652,-124.618,-40.665,178.771,5.753,149.387
C08170=1171.647,-124.368,-40.674,178.773,5.753,149.387
C08171=1171.641,-124.119,-40.683,178.775,5.753,149.386
C08172=1171.636,-123.869,-40.692,178.777,5.753,149.386
C08173=1171.631,-123.619,-40.701,178.779,5.754,149.385
C08174=1171.626,-123.369,-40.709,178.781,5.754,149.385
C08175=1171.620,-123.119,-40.718,178.783,5.754,149.384
C08176=1171.615,-122.870,-40.726,178.785,5.754,149.383
C08177=1171.609,-122.620,-40.735,178.787,5.755,149.383
C08178=1171.604,-122.370,-40.744,178.789,5.755,149.382
C08179=1171.599,-122.120,-40.753,178.792,5.755,149.382
C08180=1171.594,-121.870,-40.762,178.793,5.755,149.381
C08181=1171.588,-121.621,-40.770,178.796,5.756,149.381
C08182=1171.583,-121.371,-40.779,178.798,5.755,149.380
C08183=1171.578,-121.121,-40.788,178.800,5.756,149.379
C08184=1171.573,-120.872,-40.797,178.801,5.756,149.379
C08185=1171.567,-120.621,-40.805,178.804,5.757,149.378
C08186=1171.562,-120.371,-40.814,178.806,5.757,149.378
C08187=1171.556,-120.122,-40.823,178.808,5.757,149.377
C08188=1171.550,-119.872,-40.832,178.810,5.757,149.377
C08189=1171.545,-119.622,-40.841,178.812,5.758,149.376
C08190=1171.540,-119.372,-40.850,178.814,5.758,149.376
C08191=1171.535,-119.122,-40.859,178.816,5.758,149.375
C08192=1171.530,-118.873,-40.868,178.818,5.758,149.374
C08193=1171.524,-118.623,-40.876,178.820,5.759,149.374
C08194=1171.519,-118.374,-40.885,178.822,5.758,149.373
C08195=1171.514,-118.124,-40.894,178.824,5.759,149.373
C08196=1171.508,-117.874,-40.903,178.826,5.759,149.372
C08197=1171.502,-117.624,-40.912,178.829,5.759,149.372
C08198=1171.497,-117.374,-40.921,178.830,5.759,149.371
C08199=1171.492,-117.124,-40.930,178.833,5.760,149.370
C08200=1171.486,-116.875,-40.939,178.835,5.760,149.370
C08201=1171.481,-116.625,-40.948,178.837,5.761,149.369
C08202=1171.476,-116.375,-40.957,178.839,5.760,149.369
C08203=1171.471,-116.125,-40.965,178.841,5.761,149.368
C08204=1171.465,-115.876,-40.976,178.843,5.761,149.368
C08205=1171.460,-115.626,-40.985,178.845,5.761,149.367
C08206=1171.455,-115.376,-40.993,178.847,5.761,149.366
C08207=1171.450,-115.126,-41.002,178.850,5.762,149.366
C08208=1171.444,-114.877,-41.011,178.851,5.762,149.365
C08209=1171.439,-114.627,-41.020,178.853,5.762,149.365
C08210=1171.433,-114.377,-41.029,178.856,5.762,149.364
C08211=1171.428,-114.127,-41.038,178.858,5.763,149.364
C08212=1171.423,-113.877,-41.047,178.859,5.763,149.363
C08213=1171.417,-113.628,-41.056,178.862,5.763,149.362
C08214=1171.412,-113.377,-41.065,178.864,5.764,149.362
C08215=1171.407,-113.128,-41.075,178.866,5.763,149.361
C08216=1171.401,-112.878,-41.084,178.868,5.764,149.361
C08217=1171.396,-112.628,-41.093,178.870,5.764,149.360
C08218=1171.391,-112.379,-41.101,178.873,5.764,149.359
C08219=1171.385,-112.129,-41.111,178.874,5.764,149.359
C08220=1171.379,-111.879,-41.120,178.877,5.765,149.359
C08221=1171.374,-111.629,-41.129,178.879,5.765,149.358
C08222=1171.369,-111.380,-41.138,178.881,5.766,149.357
C08223=1171.364,-111.130,-41.148,178.883,5.765,149.357
C08224=1171.358,-110.880,-41.157,178.885,5.766,149.356
C08225=1171.353,-110.630,-41.166,178.887,5.766,149.356
C08226=1171.348,-110.380,-41.175,178.889,5.766,149.355
C08227=1171.342,-110.131,-41.185,178.891,5.766,149.354
C08228=1171.337,-109.881,-41.194,178.894,5.767,149.354
C08229=1171.332,-109.631,-41.203,178.896,5.767,149.353
C08230=1171.326,-109.381,-41.212,178.897,5.767,149.353
C08231=1171.321,-109.131,-41.221,178.900,5.768,149.352
C08232=1171.316,-108.882,-41.231,178.902,5.768,149.352
C08233=1171.311,-108.632,-41.239,178.904,5.768,149.351
C08234=1171.305,-108.382,-41.249,178.906,5.768,149.350
C08235=1171.300,-108.132,-41.258,178.908,5.769,149.350
C08236=1171.295,-107.883,-41.267,178.910,5.768,149.349
C08237=1171.289,-107.633,-41.277,178.912,5.769,149.349
C08238=1171.284,-107.383,-41.286,178.914,5.769,149.348
C08239=1171.279,-107.134,-41.295,178.917,5.770,149.347
C08240=1171.273,-106.883,-41.305,178.919,5.770,149.347
C08241=1171.268,-106.634,-41.314,178.921,5.770,149.346
C08242=1171.263,-106.384,-41.323,178.923,5.771,149.346
C08243=1171.257,-106.134,-41.333,178.925,5.770,149.345
C08244=1171.252,-105.884,-41.342,178.927,5.771,149.345
C08245=1171.247,-105.634,-41.351,178.930,5.771,149.344
C08246=1171.241,-105.385,-41.361,178.932,5.771,149.343
C08247=1171.236,-105.135,-41.370,178.933,5.771,149.343
C08248=1171.231,-104.885,-41.379,178.936,5.772,149.342
C08249=1171.225,-104.636,-41.389,178.938,5.773,149.342
C08250=1171.220,-104.386,-41.398,178.940,5.772,149.341
C08251=1171.215,-104.137,-41.407,178.942,5.773,149.341
C08252=1171.210,-103.886,-41.417,178.944,5.773,149.340
C08253=1171.204,-103.637,-41.426,178.947,5.773,149.339
C08254=1171.199,-103.387,-41.436,178.948,5.773,149.339
C08255=1171.194,-103.137,-41.445,178.951,5.774,149.338
C08256=1171.188,-102.887,-41.454,178.953,5.774,149.338
C08257=1171.183,-102.638,-41.464,178.955,5.774,149.337
C08258=1171.177,-102.366,-41.474,178.957,5.775,149.336
C08259=1171.172,-102.094,-41.484,178.960,5.774,149.336
C08260=1171.166,-101.823,-41.494,178.962,5.775,149.335
C08261=1171.160,-101.551,-41.505,178.964,5.776,149.335
C08262=1171.154,-101.301,-41.514,178.967,5.775,149.334
C08263=1171.149,-101.051,-41.524,178.969,5.776,149.333
C08264=1171.144,-100.801,-41.533,178.971,5.776,149.333
C08265=1171.139,-100.551,-41.543,178.973,5.776,149.332
C08266=1171.133,-100.301,-41.553,178.975,5.777,149.332
C08267=1171.129,-100.052,-41.562,178.977,5.777,149.331
C08268=1171.123,-99.802,-41.572,178.979,5.777,149.330
C08269=1171.118,-99.553,-41.581,178.982,5.777,149.330
C08270=1171.112,-99.302,-41.591,178.984,5.778,149.329
C08271=1171.107,-99.053,-41.600,178.986,5.778,149.329
C08272=1171.101,-98.803,-41.610,178.988,5.778,149.328
C08273=1171.096,-98.554,-41.620,178.990,5.779,149.328
C08274=1171.090,-98.304,-41.629,178.992,5.778,149.327
C08275=1171.086,-98.054,-41.639,178.994,5.779,149.326
C08276=1171.080,-97.804,-41.649,178.997,5.780,149.326
C08277=1171.075,-97.554,-41.658,178.999,5.780,149.325
C08278=1171.069,-97.304,-41.668,179.001,5.780,149.324
C08279=1171.065,-97.055,-41.677,179.003,5.780,149.324
C08280=1171.059,-96.805,-41.687,179.006,5.780,149.323
C08281=1171.054,-96.555,-41.696,179.007,5.780,149.323
C08282=1171.048,-96.306,-41.707,179.010,5.781,149.322
C08283=1171.043,-96.056,-41.715,179.012,5.782,149.322
C08284=1171.038,-95.806,-41.726,179.014,5.782,149.321
C08285=1171.032,-95.556,-41.736,179.016,5.782,149.320
C08286=1171.027,-95.306,-41.745,179.018,5.782,149.320
C08287=1171.022,-95.057,-41.755,179.021,5.782,149.319
C08288=1171.017,-94.807,-41.764,179.023,5.783,149.319
C08289=1171.011,-94.558,-41.774,179.025,5.783,149.318
C08290=1171.006,-94.308,-41.783,179.027,5.783,149.318
C08291=1171.001,-94.057,-41.794,179.029,5.783,149.317
C08292=1170.995,-93.808,-41.804,179.031,5.784,149.316
C08293=1170.990,-93.558,-41.813,179.034,5.784,149.316
C08294=1170.984,-93.308,-41.823,179.036,5.784,149.315
C08295=1170.980,-93.059,-41.833,179.038,5.785,149.314
C08296=1170.974,-92.809,-41.842,179.040,5.785,149.314
C08297=1170.969,-92.559,-41.853,179.042,5.785,149.313
C08298=1170.964,-92.310,-41.863,179.045,5.786,149.313
C08299=1170.958,-92.059,-41.872,179.046,5.786,149.312
C08300=1170.953,-91.810,-41.882,179.049,5.786,149.312
C08301=1170.947,-91.561,-41.892,179.051,5.786,149.311
C08302=1170.942,-91.310,-41.902,179.053,5.786,149.310
C08303=1170.937,-91.061,-41.911,179.056,5.787,149.310
C08304=1170.932,-90.811,-41.922,179.058,5.787,149.309
C08305=1170.926,-90.562,-41.932,179.060,5.788,149.309
C08306=1170.921,-90.312,-41.941,179.062,5.788,149.308
C08307=1170.916,-90.061,-41.951,179.064,5.788,149.307
C08308=1170.910,-89.812,-41.961,179.067,5.788,149.307
C08309=1170.905,-89.563,-41.971,179.068,5.788,149.306
C08310=1170.900,-89.312,-41.981,179.071,5.789,149.306
C08311=1170.895,-89.062,-41.991,179.073,5.790,149.305
C08312=1170.890,-88.813,-42.001,179.075,5.789,149.304
C08313=1170.884,-88.563,-42.011,179.077,5.790,149.304
C08314=1170.878,-88.314,-42.021,179.080,5.790,149.303
C08315=1170.874,-88.063,-42.030,179.082,5.790,149.303
C08316=1170.868,-87.814,-42.041,179.084,5.791,149.302
C08317=1170.863,-87.564,-42.051,179.086,5.791,149.302
C08318=1170.858,-87.315,-42.060,179.089,5.791,149.301
C08319=1170.853,-87.065,-42.071,179.091,5.792,149.300
C08320=1170.847,-86.815,-42.081,179.093,5.791,149.300
C08321=1170.841,-86.565,-42.091,179.095,5.792,149.299
C08322=1170.836,-86.316,-42.100,179.097,5.792,149.298
C08323=1170.831,-86.066,-42.111,179.099,5.793,149.298
C08324=1170.826,-85.816,-42.121,179.102,5.793,149.297
C08325=1170.821,-85.567,-42.131,179.104,5.793,149.297
C08326=1170.815,-85.317,-42.141,179.106,5.793,149.296
C08327=1170.810,-85.066,-42.151,179.109,5.794,149.296
C08328=1170.805,-84.817,-42.161,179.110,5.794,149.295
C08329=1170.800,-84.568,-42.171,179.113,5.795,149.294
C08330=1170.795,-84.317,-42.181,179.115,5.795,149.294
C08331=1170.789,-84.068,-42.191,179.117,5.795,149.293
C08332=1170.783,-83.818,-42.202,179.119,5.796,149.293
C08333=1170.778,-83.568,-42.212,179.121,5.795,149.292
C08334=1170.774,-83.319,-42.222,179.124,5.796,149.291
C08335=1170.768,-83.069,-42.232,179.126,5.796,149.291
C08336=1170.763,-82.819,-42.243,179.128,5.796,149.290
C08337=1170.757,-82.570,-42.253,179.130,5.797,149.290
C08338=1170.752,-82.320,-42.263,179.133,5.797,149.289
C08339=1170.747,-82.071,-42.273,179.135,5.797,149.288
C08340=1170.742,-81.820,-42.282,179.137,5.798,149.288
C08341=1170.736,-81.570,-42.293,179.140,5.798,149.287
C08342=1170.730,-81.321,-42.303,179.142,5.798,149.286
C08343=1170.725,-81.071,-42.313,179.144,5.799,149.286
C08344=1170.721,-80.821,-42.323,179.147,5.799,149.285
C08345=1170.715,-80.572,-42.333,179.148,5.799,149.285
C08346=1170.710,-80.322,-42.344,179.151,5.800,149.284
C08347=1170.704,-80.072,-42.354,179.153,5.800,149.284
C08348=1170.699,-79.822,-42.365,179.155,5.800,149.283
C08349=1170.694,-79.573,-42.376,179.157,5.801,149.282
C08350=1170.689,-79.323,-42.386,179.159,5.800,149.282
C08351=1170.684,-79.073,-42.396,179.162,5.801,149.281
C08352=1170.679,-78.824,-42.406,179.164,5.802,149.281
C08353=1170.673,-78.574,-42.416,179.166,5.802,149.280
C08354=1170.668,-78.324,-42.427,179.168,5.802,149.279
C08355=1170.662,-78.074,-42.437,179.171,5.803,149.279
C08356=1170.657,-77.825,-42.447,179.173,5.802,149.278
C08357=1170.652,-77.575,-42.458,179.175,5.803,149.278
C08358=1170.646,-77.325,-42.468,179.178,5.804,149.277
C08359=1170.641,-77.075,-42.479,179.179,5.804,149.276
C08360=1170.636,-76.825,-42.489,179.182,5.804,149.276
C08361=1170.630,-76.576,-42.499,179.184,5.805,149.275
C08362=1170.625,-76.305,-42.511,179.187,5.805,149.275
C08363=1170.619,-76.034,-42.522,179.189,5.805,149.274
C08364=1170.613,-75.763,-42.533,179.192,5.805,149.273
C08365=1170.608,-75.491,-42.544,179.194,5.806,149.273
C08366=1170.602,-75.242,-42.554,179.196,5.806,149.272
C08367=1170.597,-74.992,-42.566,179.198,5.806,149.271
C08368=1170.592,-74.743,-42.576,179.201,5.807,149.271
C08369=1170.587,-74.492,-42.587,179.203,5.807,149.270
C08370=1170.581,-74.243,-42.597,179.205,5.807,149.270
C08371=1170.576,-73.993,-42.607,179.207,5.808,149.269
C08372=1170.570,-73.743,-42.618,179.210,5.808,149.268
C08373=1170.565,-73.494,-42.628,179.212,5.808,149.268
C08374=1170.560,-73.244,-42.639,179.214,5.809,149.267
C08375=1170.555,-72.994,-42.649,179.217,5.809,149.267
C08376=1170.550,-72.744,-42.660,179.219,5.810,149.266
C08377=1170.544,-72.495,-42.671,179.221,5.809,149.265
C08378=1170.539,-72.245,-42.681,179.223,5.810,149.265
C08379=1170.534,-71.995,-42.692,179.226,5.811,149.264
C08380=1170.529,-71.745,-42.702,179.227,5.811,149.264
C08381=1170.523,-71.496,-42.713,179.230,5.811,149.263
C08382=1170.518,-71.247,-42.723,179.232,5.812,149.262
C08383=1170.513,-70.996,-42.734,179.234,5.811,149.262
C08384=1170.507,-70.747,-42.744,179.237,5.812,149.261
C08385=1170.503,-70.497,-42.755,179.239,5.813,149.261
C08386=1170.497,-70.248,-42.766,179.241,5.812,149.260
C08387=1170.492,-69.997,-42.776,179.243,5.813,149.259
C08388=1170.487,-69.749,-42.787,179.246,5.813,149.259
C08389=1170.482,-69.498,-42.798,179.248,5.814,149.258
C08390=1170.476,-69.249,-42.808,179.250,5.814,149.257
C08391=1170.471,-68.998,-42.818,179.253,5.815,149.257
C08392=1170.465,-68.749,-42.830,179.255,5.815,149.256
C08393=1170.460,-68.499,-42.840,179.257,5.815,149.256
C08394=1170.454,-68.249,-42.851,179.260,5.815,149.255
C08395=1170.450,-68.000,-42.862,179.262,5.816,149.255
C08396=1170.444,-67.750,-42.872,179.264,5.816,149.254
C08397=1170.439,-67.501,-42.883,179.266,5.816,149.253
C08398=1170.434,-67.251,-42.894,179.269,5.817,149.253
C08399=1170.429,-67.001,-42.904,179.271,5.817,149.252
C08400=1170.424,-66.752,-42.915,179.273,5.817,149.252
C08401=1170.418,-66.501,-42.926,179.276,5.818,149.251
C08402=1170.413,-66.252,-42.938,179.278,5.819,149.250
C08403=1170.408,-66.002,-42.948,179.280,5.818,149.250
C08404=1170.403,-65.752,-42.958,179.282,5.819,149.249
C08405=1170.397,-65.503,-42.969,179.285,5.819,149.248
C08406=1170.392,-65.253,-42.980,179.287,5.820,149.248
C08407=1170.387,-65.004,-42.991,179.289,5.820,149.247
C08408=1170.381,-64.753,-43.002,179.292,5.820,149.247
C08409=1170.376,-64.504,-43.013,179.294,5.821,149.246
C08410=1170.371,-64.254,-43.023,179.296,5.821,149.245
C08411=1170.366,-64.005,-43.035,179.298,5.821,149.245
C08412=1170.361,-63.755,-43.045,179.301,5.822,149.244
C08413=1170.356,-63.505,-43.056,179.303,5.823,149.244
C08414=1170.350,-63.256,-43.067,179.305,5.822,149.243
C08415=1170.345,-63.006,-43.078,179.307,5.823,149.243
C08416=1170.340,-62.756,-43.089,179.310,5.823,149.242
C08417=1170.335,-62.507,-43.100,179.313,5.824,149.241
C08418=1170.329,-62.256,-43.111,179.314,5.824,149.241
C08419=1170.324,-62.007,-43.122,179.317,5.824,149.240
C08420=1170.319,-61.757,-43.133,179.319,5.825,149.239
C08421=1170.314,-61.507,-43.144,179.321,5.825,149.239
C08422=1170.308,-61.258,-43.154,179.323,5.826,149.238
C08423=1170.303,-61.008,-43.166,179.326,5.826,149.238
C08424=1170.297,-60.758,-43.176,179.329,5.826,149.237
C08425=1170.293,-60.509,-43.187,179.330,5.826,149.236
C08426=1170.288,-60.259,-43.199,179.333,5.827,149.236
C08427=1170.282,-60.009,-43.210,179.335,5.828,149.235
C08428=1170.277,-59.760,-43.221,179.338,5.828,149.235
C08429=1170.272,-59.509,-43.231,179.339,5.828,149.234
C08430=1170.267,-59.260,-43.242,179.342,5.828,149.233
C08431=1170.261,-59.011,-43.254,179.345,5.829,149.233
C08432=1170.256,-58.760,-43.265,179.347,5.830,149.232
C08433=1170.251,-58.511,-43.276,179.349,5.829,149.231
C08434=1170.245,-58.261,-43.287,179.351,5.830,149.231
C08435=1170.240,-58.012,-43.298,179.354,5.830,149.230
C08436=1170.235,-57.762,-43.309,179.356,5.831,149.230
C08437=1170.229,-57.512,-43.320,179.358,5.831,149.229
C08438=1170.224,-57.263,-43.331,179.361,5.831,149.228
C08439=1170.219,-57.013,-43.342,179.363,5.832,149.228
C08440=1170.214,-56.763,-43.353,179.366,5.832,149.227
C08441=1170.209,-56.513,-43.365,179.367,5.832,149.227
C08442=1170.204,-56.264,-43.376,179.370,5.833,149.226
C08443=1170.199,-56.014,-43.387,179.372,5.834,149.226
C08444=1170.193,-55.764,-43.398,179.375,5.834,149.225
C08445=1170.188,-55.515,-43.409,179.377,5.834,149.224
C08446=1170.183,-55.265,-43.421,179.379,5.834,149.224
C08447=1170.178,-55.015,-43.432,179.382,5.835,149.223
C08448=1170.172,-54.766,-43.443,179.384,5.836,149.222
C08449=1170.167,-54.516,-43.455,179.386,5.835,149.222
C08450=1170.162,-54.266,-43.466,179.388,5.836,149.221
C08451=1170.157,-54.017,-43.477,179.391,5.837,149.221
C08452=1170.151,-53.767,-43.488,179.393,5.837,149.220
C08453=1170.146,-53.517,-43.499,179.396,5.838,149.219
C08454=1170.141,-53.267,-43.511,179.398,5.837,149.219
C08455=1170.136,-53.018,-43.522,179.400,5.838,149.218
C08456=1170.131,-52.768,-43.533,179.402,5.839,149.218
C08457=1170.125,-52.518,-43.544,179.405,5.839,149.217
C08458=1170.121,-52.268,-43.556,179.407,5.839,149.216
C08459=1170.115,-52.019,-43.567,179.409,5.839,149.216
C08460=1170.110,-51.770,-43.579,179.412,5.840,149.215
C08461=1170.104,-51.520,-43.590,179.414,5.841,149.214
C08462=1170.099,-51.269,-43.601,179.416,5.841,149.214
C08463=1170.094,-51.021,-43.612,179.418,5.841,149.213
C08464=1170.089,-50.771,-43.624,179.421,5.841,149.213
C08465=1170.084,-50.521,-43.635,179.423,5.842,149.212
C08466=1170.078,-50.250,-43.647,179.426,5.843,149.211
C08467=1170.072,-49.980,-43.660,179.429,5.843,149.211
C08468=1170.067,-49.709,-43.672,179.431,5.844,149.210
C08469=1170.061,-49.440,-43.685,179.434,5.844,149.210
C08470=1170.056,-49.190,-43.697,179.436,5.844,149.209
C08471=1170.051,-48.940,-43.708,179.438,5.845,149.208
C08472=1170.045,-48.690,-43.719,179.440,5.845,149.208
C08473=1170.040,-48.440,-43.730,179.443,5.846,149.207
C08474=1170.034,-48.191,-43.742,179.445,5.846,149.206
C08475=1170.030,-47.941,-43.753,179.447,5.846,149.206
C08476=1170.024,-47.691,-43.765,179.450,5.847,149.205
C08477=1170.020,-47.442,-43.776,179.452,5.847,149.205
C08478=1170.014,-47.192,-43.788,179.455,5.848,149.204
C08479=1170.009,-46.943,-43.799,179.457,5.848,149.203
C08480=1170.003,-46.693,-43.811,179.459,5.848,149.203
C08481=1169.999,-46.443,-43.822,179.461,5.849,149.202
C08482=1169.993,-46.193,-43.834,179.464,5.849,149.202
C08483=1169.988,-45.943,-43.846,179.467,5.850,149.201
C08484=1169.983,-45.694,-43.857,179.469,5.851,149.200
C08485=1169.977,-45.444,-43.869,179.471,5.850,149.200
C08486=1169.972,-45.195,-43.880,179.473,5.851,149.199
C08487=1169.967,-44.945,-43.892,179.476,5.851,149.198
C08488=1169.962,-44.695,-43.903,179.478,5.852,149.198
C08489=1169.957,-44.445,-43.915,179.481,5.853,149.197
C08490=1169.951,-44.195,-43.927,179.483,5.852,149.197
C08491=1169.946,-43.946,-43.938,179.485,5.853,149.196
C08492=1169.941,-43.696,-43.950,179.488,5.853,149.195
C08493=1169.936,-43.447,-43.962,179.490,5.854,149.195
C08494=1169.931,-43.198,-43.974,179.492,5.855,149.194
C08495=1169.926,-42.948,-43.986,179.495,5.855,149.194
C08496=1169.921,-42.698,-43.997,179.497,5.855,149.193
C08497=1169.915,-42.448,-44.009,179.499,5.856,149.192
C08498=1169.910,-42.198,-44.021,179.502,5.856,149.192
C08499=1169.905,-41.949,-44.032,179.504,5.857,149.191
C08500=1169.899,-41.699,-44.044,179.507,5.857,149.190
C08501=1169.894,-41.450,-44.056,179.509,5.858,149.190
C08502=1169.889,-41.200,-44.068,179.511,5.858,149.189
C08503=1169.884,-40.950,-44.079,179.513,5.858,149.189
C08504=1169.879,-40.700,-44.091,179.516,5.859,149.188
C08505=1169.874,-40.451,-44.103,179.519,5.859,149.187
C08506=1169.868,-40.201,-44.115,179.521,5.860,149.187
C08507=1169.863,-39.952,-44.127,179.523,5.861,149.186
C08508=1169.859,-39.702,-44.138,179.525,5.861,149.186
C08509=1169.853,-39.452,-44.150,179.528,5.861,149.185
C08510=1169.847,-39.203,-44.162,179.530,5.861,149.184
C08511=1169.842,-38.953,-44.174,179.533,5.862,149.184
C08512=1169.837,-38.704,-44.186,179.535,5.863,149.183
C08513=1169.832,-38.454,-44.198,179.537,5.863,149.183
C08514=1169.826,-38.204,-44.209,179.539,5.863,149.182
C08515=1169.821,-37.954,-44.221,179.542,5.863,149.181
C08516=1169.817,-37.705,-44.233,179.544,5.864,149.181
C08517=1169.811,-37.455,-44.245,179.547,5.865,149.180
C08518=1169.806,-37.205,-44.257,179.549,5.866,149.180
C08519=1169.800,-36.955,-44.269,179.552,5.866,149.179
C08520=1169.796,-36.706,-44.281,179.554,5.866,149.178
C08521=1169.791,-36.456,-44.293,179.556,5.866,149.178
C08522=1169.785,-36.206,-44.305,179.559,5.867,149.177
C08523=1169.780,-35.957,-44.317,179.561,5.868,149.177
C08524=1169.775,-35.707,-44.329,179.564,5.868,149.176
C08525=1169.770,-35.457,-44.341,179.566,5.869,149.175
C08526=1169.765,-35.208,-44.353,179.568,5.869,149.175
C08527=1169.759,-34.958,-44.365,179.570,5.869,149.174
C08528=1169.754,-34.708,-44.377,179.573,5.870,149.174
C08529=1169.750,-34.459,-44.389,179.575,5.870,149.173
C08530=1169.744,-34.209,-44.401,179.578,5.871,149.172
C08531=1169.739,-33.959,-44.413,179.580,5.871,149.172
C08532=1169.734,-33.710,-44.425,179.583,5.872,149.171
C08533=1169.728,-33.460,-44.437,179.586,5.872,149.170
C08534=1169.723,-33.210,-44.449,179.588,5.873,149.170
C08535=1169.718,-32.961,-44.462,179.590,5.873,149.169
C08536=1169.713,-32.711,-44.473,179.592,5.874,149.169
C08537=1169.708,-32.462,-44.486,179.595,5.874,149.168
C08538=1169.702,-32.212,-44.497,179.597,5.874,149.167
C08539=1169.697,-31.963,-44.510,179.599,5.875,149.167
C08540=1169.692,-31.713,-44.522,179.602,5.876,149.166
C08541=1169.686,-31.463,-44.534,179.604,5.876,149.166
C08542=1169.681,-31.213,-44.546,179.607,5.877,149.165
C08543=1169.677,-30.964,-44.558,179.609,5.877,149.164
C08544=1169.671,-30.714,-44.570,179.611,5.877,149.164
C08545=1169.666,-30.465,-44.582,179.614,5.878,149.163
C08546=1169.661,-30.215,-44.595,179.616,5.879,149.163
C08547=1169.655,-29.965,-44.607,179.619,5.879,149.162
C08548=1169.650,-29.716,-44.619,179.621,5.879,149.161
C08549=1169.645,-29.466,-44.631,179.624,5.880,149.161
C08550=1169.640,-29.216,-44.644,179.626,5.881,149.160
C08551=1169.635,-28.966,-44.656,179.628,5.881,149.160
C08552=1169.630,-28.717,-44.669,179.630,5.881,149.159
C08553=1169.624,-28.467,-44.681,179.633,5.882,149.158
C08554=1169.619,-28.217,-44.693,179.635,5.882,149.158
C08555=1169.614,-27.968,-44.706,179.638,5.883,149.157
C08556=1169.609,-27.718,-44.718,179.641,5.883,149.156
C08557=1169.604,-27.469,-44.730,179.643,5.884,149.156
C08558=1169.598,-27.219,-44.742,179.645,5.885,149.155
C08559=1169.594,-26.970,-44.754,179.648,5.885,149.155
C08560=1169.589,-26.719,-44.766,179.650,5.886,149.154
C08561=1169.584,-26.470,-44.779,179.652,5.885,149.153
C08562=1169.579,-26.221,-44.792,179.655,5.886,149.153
C08563=1169.573,-25.971,-44.803,179.657,5.887,149.152
C08564=1169.568,-25.721,-44.816,179.659,5.887,149.152
C08565=1169.563,-25.472,-44.829,179.662,5.888,149.151
C08566=1169.558,-25.222,-44.841,179.665,5.888,149.150
C08567=1169.552,-24.973,-44.853,179.667,5.889,149.150
C08568=1169.547,-24.723,-44.867,179.670,5.890,149.149
C08569=1169.542,-24.473,-44.879,179.672,5.890,149.149
C08570=1169.536,-24.204,-44.892,179.674,5.891,149.148
C08571=1169.531,-23.933,-44.905,179.677,5.891,149.147
C08572=1169.525,-23.663,-44.919,179.680,5.892,149.147
C08573=1169.519,-23.394,-44.932,179.682,5.892,149.146
C08574=1169.515,-23.144,-44.945,179.685,5.893,149.145
C08575=1169.510,-22.894,-44.957,179.687,5.893,149.145
C08576=1169.504,-22.645,-44.970,179.690,5.894,149.144
C08577=1169.499,-22.396,-44.982,179.692,5.895,149.143
C08578=1169.494,-22.146,-44.994,179.695,5.895,149.143
C08579=1169.489,-21.896,-45.007,179.697,5.896,149.142
C08580=1169.483,-21.646,-45.021,179.699,5.896,149.142
C08581=1169.478,-21.397,-45.033,179.702,5.896,149.141
C08582=1169.473,-21.147,-45.045,179.704,5.897,149.140
C08583=1169.468,-20.897,-45.058,179.706,5.897,149.140
C08584=1169.463,-20.648,-45.070,179.709,5.898,149.139
C08585=1169.458,-20.398,-45.083,179.711,5.899,149.139
C08586=1169.453,-20.149,-45.096,179.714,5.899,149.138
C08587=1169.448,-19.899,-45.108,179.716,5.900,149.137
C08588=1169.442,-19.649,-45.121,179.719,5.900,149.137
C08589=1169.437,-19.400,-45.133,179.721,5.901,149.136
C08590=1169.432,-19.150,-45.146,179.724,5.902,149.136
C08591=1169.427,-18.901,-45.159,179.726,5.902,149.135
C08592=1169.422,-18.651,-45.172,179.728,5.903,149.134
C08593=1169.416,-18.401,-45.184,179.731,5.903,149.134
C08594=1169.411,-18.151,-45.197,179.734,5.904,149.133
C08595=1169.406,-17.902,-45.210,179.736,5.905,149.133
C08596=1169.401,-17.652,-45.222,179.738,5.904,149.132
C08597=1169.396,-17.403,-45.235,179.740,5.905,149.131
C08598=1169.391,-17.153,-45.248,179.743,5.905,149.131
C08599=1169.385,-16.903,-45.261,179.746,5.906,149.130
C08600=1169.380,-16.654,-45.274,179.748,5.907,149.130
C08601=1169.375,-16.405,-45.286,179.750,5.907,149.129
C08602=1169.371,-16.155,-45.299,179.753,5.908,149.128
C08603=1169.365,-15.905,-45.311,179.755,5.908,149.128
C08604=1169.359,-15.655,-45.324,179.758,5.909,149.127
C08605=1169.354,-15.406,-45.337,179.760,5.910,149.127
C08606=1169.350,-15.156,-45.350,179.763,5.910,149.126
C08607=1169.345,-14.906,-45.362,179.765,5.911,149.125
C08608=1169.339,-14.657,-45.376,179.768,5.911,149.125
C08609=1169.334,-14.407,-45.389,179.770,5.912,149.124
C08610=1169.329,-14.158,-45.401,179.772,5.913,149.124
C08611=1169.323,-13.908,-45.414,179.775,5.913,149.123
C08612=1169.319,-13.658,-45.427,179.778,5.914,149.122
C08613=1169.314,-13.409,-45.440,179.780,5.914,149.122
C08614=1169.308,-13.159,-45.453,179.783,5.915,149.121
C08615=1169.303,-12.909,-45.466,179.785,5.915,149.120
C08616=1169.298,-12.660,-45.479,179.787,5.916,149.120
C08617=1169.293,-12.411,-45.492,179.790,5.917,149.119
C08618=1169.288,-12.161,-45.506,179.792,5.917,149.119
C08619=1169.283,-11.911,-45.518,179.795,5.918,149.118
C08620=1169.278,-11.662,-45.531,179.798,5.918,149.117
C08621=1169.272,-11.412,-45.544,179.800,5.919,149.117
C08622=1169.267,-11.162,-45.557,179.802,5.920,149.116
C08623=1169.262,-10.913,-45.570,179.805,5.920,149.116
C08624=1169.257,-10.663,-45.583,179.807,5.921,149.115
C08625=1169.252,-10.413,-45.596,179.810,5.921,149.114
C08626=1169.247,-10.164,-45.608,179.812,5.922,149.114
C08627=1169.242,-9.914,-45.623,179.815,5.923,149.113
C08628=1169.237,-9.665,-45.635,179.817,5.923,149.113
C08629=1169.231,-9.416,-45.648,179.819,5.924,149.112
C08630=1169.226,-9.165,-45.661,179.822,5.924,149.111
C08631=1169.221,-8.916,-45.674,179.824,5.925,149.111
C08632=1169.216,-8.666,-45.688,179.827,5.926,149.110
C08633=1169.211,-8.417,-45.701,179.830,5.926,149.109
C08634=1169.206,-8.168,-45.713,179.832,5.927,149.109
C08635=1169.201,-7.917,-45.727,179.834,5.927,149.108
C08636=1169.196,-7.668,-45.740,179.837,5.928,149.108
C08637=1169.190,-7.418,-45.753,179.839,5.929,149.107
C08638=1169.185,-7.169,-45.767,179.842,5.929,149.106
C08639=1169.180,-6.919,-45.780,179.844,5.930,149.106
C08640=1169.175,-6.669,-45.793,179.847,5.930,149.105
C08641=1169.170,-6.420,-45.805,179.849,5.931,149.105
C08642=1169.165,-6.170,-45.820,179.852,5.932,149.104
C08643=1169.160,-5.921,-45.832,179.854,5.932,149.103
C08644=1169.155,-5.671,-45.846,179.856,5.933,149.103
C08645=1169.149,-5.421,-45.858,179.859,5.933,149.102
C08646=1169.145,-5.172,-45.873,179.862,5.934,149.102
C08647=1169.139,-4.922,-45.885,179.864,5.935,149.101
C08648=1169.134,-4.673,-45.898,179.867,5.935,149.100
C08649=1169.129,-4.423,-45.912,179.869,5.936,149.100
C08650=1169.123,-4.174,-45.925,179.871,5.936,149.099
C08651=1169.119,-3.924,-45.938,179.874,5.937,149.099
C08652=1169.113,-3.675,-45.952,179.876,5.938,149.098
C08653=1169.109,-3.425,-45.965,179.879,5.938,149.097
C08654=1169.103,-3.175,-45.978,179.881,5.939,149.097
C08655=1169.099,-2.926,-45.992,179.884,5.939,149.096
C08656=1169.093,-2.676,-46.005,179.886,5.940,149.096
C08657=1169.089,-2.427,-46.019,179.889,5.941,149.095
C08658=1169.083,-2.177,-46.032,179.891,5.941,149.094
C08659=1169.078,-1.927,-46.046,179.893,5.942,149.094
C08660=1169.073,-1.678,-46.059,179.896,5.942,149.093
C08661=1169.067,-1.428,-46.073,179.899,5.943,149.093
C08662=1169.063,-1.179,-46.086,179.901,5.944,149.092
C08663=1169.057,-0.929,-46.099,179.904,5.944,149.091
C08664=1169.052,-0.679,-46.112,179.906,5.945,149.091
C08665=1169.047,-0.430,-46.126,179.908,5.945,149.090
C08666=1169.041,-0.180,-46.139,179.911,5.946,149.090
C08667=1169.037,0.070,-46.153,179.913,5.947,149.089
C08668=1169.031,0.319,-46.166,179.916,5.947,149.088
C08669=1169.027,0.569,-46.180,179.918,5.948,149.088
C08670=1169.021,0.818,-46.193,179.921,5.948,149.087
C08671=1169.016,1.068,-46.208,179.923,5.949,149.087
C08672=1169.011,1.317,-46.220,179.926,5.951,149.086
C08673=1169.006,1.567,-46.234,179.929,5.951,149.085
C08674=1169.001,1.836,-46.249,179.931,5.951,149.085
C08675=1168.995,2.106,-46.263,179.934,5.952,149.084
C08676=1168.990,2.375,-46.278,179.936,5.953,149.084
C08677=1168.984,2.644,-46.293,179.939,5.953,149.083
C08678=1168.979,2.893,-46.307,179.942,5.954,149.082
C08679=1168.974,3.144,-46.320,179.944,5.955,149.082
C08680=1168.969,3.393,-46.334,179.947,5.956,149.081
C08681=1168.963,3.643,-46.347,179.950,5.956,149.080
C08682=1168.959,3.892,-46.361,179.952,5.957,149.080
C08683=1168.954,4.141,-46.375,179.954,5.957,149.079
C08684=1168.948,4.391,-46.388,179.957,5.958,149.079
C08685=1168.943,4.641,-46.402,179.959,5.959,149.078
C08686=1168.938,4.890,-46.415,179.962,5.959,149.077
C08687=1168.933,5.140,-46.429,179.964,5.960,149.077
C08688=1168.928,5.389,-46.443,179.967,5.961,149.076
C08689=1168.923,5.639,-46.457,179.969,5.961,149.076
C08690=1168.918,5.889,-46.470,179.972,5.962,149.075
C08691=1168.913,6.138,-46.484,179.974,5.962,149.074
C08692=1168.908,6.388,-46.498,179.977,5.964,149.074
C08693=1168.902,6.637,-46.512,179.980,5.964,149.073
C08694=1168.898,6.886,-46.526,179.982,5.965,149.073
C08695=1168.893,7.137,-46.539,179.984,5.966,149.072
C08696=1168.887,7.386,-46.553,179.987,5.966,149.071
C08697=1168.882,7.636,-46.567,179.989,5.967,149.071
C08698=1168.877,7.885,-46.582,179.992,5.967,149.070
C08699=1168.872,8.135,-46.594,179.995,5.968,149.070
C08700=1168.867,8.384,-46.608,179.997,5.969,149.069
C08701=1168.862,8.634,-46.623,179.999,5.969,149.068
C08702=1168.856,8.883,-46.637,-179.998,5.970,149.068
C08703=1168.851,9.133,-46.650,-179.996,5.971,149.067
C08704=1168.847,9.383,-46.664,-179.993,5.972,149.067
C08705=1168.841,9.632,-46.678,-179.990,5.973,149.066
C08706=1168.836,9.881,-46.692,-179.988,5.973,149.065
C08707=1168.832,10.131,-46.706,-179.986,5.974,149.065
C08708=1168.826,10.381,-46.720,-179.983,5.974,149.064
C08709=1168.821,10.631,-46.734,-179.980,5.975,149.064
C08710=1168.817,10.880,-46.748,-179.978,5.976,149.063
C08711=1168.811,11.129,-46.761,-179.975,5.976,149.063
C08712=1168.806,11.379,-46.776,-179.973,5.977,149.062
C08713=1168.801,11.628,-46.790,-179.970,5.978,149.061
C08714=1168.796,11.879,-46.804,-179.968,5.979,149.061
C08715=1168.790,12.128,-46.817,-179.965,5.980,149.060
C08716=1168.785,12.377,-46.832,-179.963,5.980,149.060
C08717=1168.780,12.627,-46.846,-179.960,5.981,149.059
C08718=1168.775,12.876,-46.860,-179.958,5.981,149.058
C08719=1168.771,13.125,-46.874,-179.956,5.982,149.058
C08720=1168.766,13.375,-46.888,-179.953,5.983,149.057
C08721=1168.761,13.625,-46.902,-179.950,5.983,149.057
C08722=1168.755,13.874,-46.916,-179.948,5.985,149.056
C08723=1168.750,14.124,-46.930,-179.945,5.985,149.055
C08724=1168.745,14.373,-46.945,-179.943,5.986,149.055
C08725=1168.740,14.624,-46.958,-179.940,5.987,149.054
C08726=1168.734,14.873,-46.972,-179.937,5.987,149.054
C08727=1168.729,15.122,-46.986,-179.935,5.988,149.053
C08728=1168.724,15.372,-47.001,-179.933,5.988,149.052
C08729=1168.719,15.622,-47.015,-179.930,5.989,149.052
C08730=1168.715,15.872,-47.029,-179.927,5.990,149.051
C08731=1168.709,16.121,-47.043,-179.925,5.991,149.051
C08732=1168.704,16.370,-47.057,-179.922,5.992,149.050
C08733=1168.699,16.620,-47.072,-179.920,5.992,149.050
C08734=1168.694,16.869,-47.087,-179.918,5.993,149.049
C08735=1168.689,17.118,-47.101,-179.915,5.994,149.048
C08736=1168.684,17.368,-47.115,-179.912,5.994,149.048
C08737=1168.679,17.617,-47.129,-179.910,5.996,149.047
C08738=1168.674,17.867,-47.143,-179.907,5.996,149.047
C08739=1168.669,18.117,-47.158,-179.905,5.997,149.046
C08740=1168.664,18.367,-47.172,-179.902,5.997,149.045
C08741=1168.659,18.616,-47.186,-179.900,5.998,149.045
C08742=1168.654,18.865,-47.200,-179.897,5.999,149.044
C08743=1168.649,19.115,-47.214,-179.895,5.999,149.044
C08744=1168.644,19.365,-47.229,-179.892,6.001,149.043
C08745=1168.639,19.614,-47.244,-179.889,6.001,149.042
C08746=1168.633,19.863,-47.258,-179.887,6.002,149.042
C08747=1168.628,20.113,-47.272,-179.884,6.003,149.041
C08748=1168.623,20.363,-47.287,-179.882,6.003,149.041
C08749=1168.618,20.612,-47.301,-179.880,6.004,149.040
C08750=1168.613,20.862,-47.315,-179.876,6.005,149.040
C08751=1168.608,21.111,-47.330,-179.874,6.006,149.039
C08752=1168.603,21.361,-47.345,-179.871,6.007,149.038
C08753=1168.598,21.610,-47.358,-179.869,6.007,149.038
C08754=1168.593,21.860,-47.373,-179.867,6.008,149.037
C08755=1168.588,22.109,-47.387,-179.864,6.008,149.037
C08756=1168.582,22.359,-47.403,-179.861,6.010,149.036
C08757=1168.577,22.608,-47.417,-179.859,6.011,149.035
C08758=1168.573,22.858,-47.431,-179.856,6.011,149.035
C08759=1168.568,23.108,-47.445,-179.854,6.012,149.034
C08760=1168.563,23.357,-47.460,-179.851,6.012,149.034
C08761=1168.558,23.607,-47.475,-179.848,6.014,149.033
C08762=1168.552,23.856,-47.489,-179.846,6.014,149.032
C08763=1168.547,24.106,-47.504,-179.844,6.015,149.032
C08764=1168.542,24.355,-47.519,-179.841,6.016,149.031
C08765=1168.537,24.604,-47.533,-179.839,6.017,149.031
C08766=1168.532,24.854,-47.547,-179.836,6.017,149.030
C08767=1168.528,25.103,-47.562,-179.833,6.018,149.030
C08768=1168.522,25.353,-47.577,-179.831,6.019,149.029
C08769=1168.517,25.603,-47.591,-179.828,6.020,149.028
C08770=1168.512,25.852,-47.606,-179.826,6.021,149.028
C08771=1168.507,26.102,-47.620,-179.823,6.021,149.027
C08772=1168.502,26.352,-47.635,-179.821,6.023,149.027
C08773=1168.497,26.601,-47.650,-179.818,6.023,149.026
C08774=1168.492,26.851,-47.665,-179.815,6.024,149.025
C08775=1168.487,27.100,-47.680,-179.813,6.025,149.025
C08776=1168.482,27.350,-47.694,-179.810,6.025,149.024
C08777=1168.477,27.599,-47.709,-179.808,6.027,149.024
C08778=1168.471,27.867,-47.724,-179.805,6.027,149.023
C08779=1168.465,28.137,-47.740,-179.802,6.028,149.023
C08780=1168.460,28.405,-47.756,-179.799,6.029,149.022
C08781=1168.455,28.674,-47.772,-179.797,6.030,149.021
C08782=1168.449,28.924,-47.787,-179.794,6.030,149.021
C08783=1168.444,29.173,-47.802,-179.791,6.032,149.020
C08784=1168.440,29.422,-47.817,-179.789,6.032,149.020
C08785=1168.434,29.672,-47.832,-179.786,6.033,149.019
C08786=1168.430,29.921,-47.847,-179.784,6.034,149.018
C08787=1168.425,30.171,-47.861,-179.782,6.034,149.018
C08788=1168.419,30.421,-47.876,-179.779,6.036,149.017
C08789=1168.414,30.670,-47.891,-179.776,6.036,149.017
C08790=1168.410,30.919,-47.906,-179.774,6.037,149.016
C08791=1168.404,31.169,-47.921,-179.771,6.038,149.016
C08792=1168.399,31.419,-47.936,-179.768,6.039,149.015
C08793=1168.394,31.668,-47.950,-179.766,6.040,149.014
C08794=1168.389,31.918,-47.966,-179.763,6.040,149.014
C08795=1168.385,32.167,-47.981,-179.761,6.041,149.013
C08796=1168.379,32.417,-47.996,-179.758,6.042,149.013
C08797=1168.374,32.667,-48.011,-179.756,6.043,149.012
C08798=1168.370,32.916,-48.025,-179.753,6.044,149.011
C08799=1168.364,33.166,-48.040,-179.750,6.044,149.011
C08800=1168.359,33.415,-48.055,-179.748,6.045,149.010
C08801=1168.354,33.665,-48.070,-179.745,6.046,149.010
C08802=1168.349,33.914,-48.085,-179.743,6.047,149.009
C08803=1168.345,34.163,-48.100,-179.740,6.048,149.009
C08804=1168.339,34.413,-48.115,-179.738,6.049,149.008
C08805=1168.334,34.662,-48.130,-179.735,6.050,149.007
C08806=1168.329,34.911,-48.146,-179.733,6.051,149.007
C08807=1168.324,35.161,-48.160,-179.730,6.051,149.006
C08808=1168.318,35.411,-48.176,-179.727,6.052,149.006
C08809=1168.314,35.660,-48.191,-179.725,6.053,149.005
C08810=1168.309,35.910,-48.206,-179.722,6.054,149.005
C08811=1168.304,36.159,-48.221,-179.720,6.055,149.004
C08812=1168.299,36.409,-48.236,-179.717,6.055,149.003
C08813=1168.294,36.659,-48.251,-179.714,6.057,149.003
C08814=1168.288,36.908,-48.266,-179.712,6.057,149.002
C08815=1168.284,37.157,-48.281,-179.710,6.058,149.002
C08816=1168.278,37.406,-48.297,-179.707,6.059,149.001
C08817=1168.274,37.656,-48.312,-179.704,6.060,149.001
C08818=1168.269,37.906,-48.327,-179.702,6.061,149.000
C08819=1168.264,38.155,-48.342,-179.699,6.061,148.999
C08820=1168.259,38.405,-48.358,-179.696,6.063,148.999
C08821=1168.254,38.654,-48.373,-179.694,6.063,148.998
C08822=1168.248,38.903,-48.388,-179.691,6.064,148.998
C08823=1168.243,39.153,-48.403,-179.689,6.065,148.997
C08824=1168.239,39.403,-48.419,-179.686,6.066,148.997
C08825=1168.233,39.653,-48.434,-179.683,6.067,148.996
C08826=1168.229,39.902,-48.449,-179.681,6.068,148.996
C08827=1168.223,40.151,-48.465,-179.679,6.068,148.995
C08828=1168.219,40.400,-48.480,-179.676,6.070,148.994
C08829=1168.213,40.650,-48.495,-179.673,6.070,148.994
C08830=1168.208,40.900,-48.511,-179.671,6.071,148.993
C08831=1168.204,41.149,-48.526,-179.668,6.073,148.993
C08832=1168.198,41.399,-48.541,-179.665,6.073,148.992
C08833=1168.193,41.648,-48.557,-179.663,6.074,148.992
C08834=1168.188,41.897,-48.572,-179.660,6.074,148.991
C08835=1168.183,42.147,-48.588,-179.658,6.076,148.990
C08836=1168.179,42.396,-48.603,-179.655,6.077,148.990
C08837=1168.173,42.646,-48.618,-179.653,6.077,148.989
C08838=1168.168,42.895,-48.634,-179.650,6.079,148.989
C08839=1168.163,43.144,-48.649,-179.647,6.080,148.988
C08840=1168.158,43.394,-48.665,-179.645,6.080,148.987
C08841=1168.153,43.644,-48.680,-179.642,6.082,148.987
C08842=1168.148,43.893,-48.695,-179.639,6.082,148.986
C08843=1168.143,44.142,-48.711,-179.637,6.083,148.986
C08844=1168.138,44.392,-48.727,-179.635,6.084,148.985
C08845=1168.134,44.641,-48.742,-179.631,6.085,148.985
C08846=1168.128,44.891,-48.757,-179.629,6.086,148.984
C08847=1168.123,45.140,-48.773,-179.627,6.086,148.983
C08848=1168.118,45.390,-48.789,-179.624,6.088,148.983
C08849=1168.113,45.639,-48.804,-179.621,6.088,148.982
C08850=1168.108,45.889,-48.820,-179.619,6.089,148.982
C08851=1168.103,46.138,-48.835,-179.616,6.091,148.981
C08852=1168.098,46.388,-48.851,-179.614,6.091,148.981
C08853=1168.093,46.637,-48.866,-179.611,6.092,148.980
C08854=1168.088,46.887,-48.882,-179.608,6.094,148.980
C08855=1168.083,47.136,-48.898,-179.606,6.094,148.979
C08856=1168.078,47.386,-48.914,-179.603,6.095,148.979
C08857=1168.073,47.635,-48.929,-179.600,6.096,148.978
C08858=1168.068,47.885,-48.945,-179.598,6.097,148.977
C08859=1168.063,48.134,-48.960,-179.595,6.098,148.977
C08860=1168.058,48.384,-48.976,-179.593,6.099,148.976
C08861=1168.053,48.632,-48.992,-179.590,6.100,148.976
C08862=1168.049,48.882,-49.008,-179.588,6.101,148.975
C08863=1168.043,49.132,-49.023,-179.585,6.102,148.975
C08864=1168.038,49.381,-49.039,-179.582,6.103,148.974
C08865=1168.033,49.631,-49.055,-179.580,6.103,148.973
C08866=1168.028,49.880,-49.071,-179.577,6.105,148.973
C08867=1168.023,50.129,-49.086,-179.575,6.106,148.972
C08868=1168.019,50.379,-49.102,-179.572,6.106,148.972
C08869=1168.013,50.629,-49.118,-179.569,6.108,148.971
C08870=1168.009,50.878,-49.134,-179.566,6.108,148.971
C08871=1168.003,51.128,-49.150,-179.564,6.109,148.970
C08872=1167.998,51.377,-49.166,-179.561,6.110,148.969
C08873=1167.993,51.627,-49.182,-179.559,6.111,148.969
C08874=1167.989,51.875,-49.197,-179.556,6.112,148.968
C08875=1167.983,52.125,-49.213,-179.554,6.113,148.968
C08876=1167.979,52.375,-49.229,-179.551,6.114,148.967
C08877=1167.973,52.624,-49.245,-179.549,6.115,148.967
C08878=1167.969,52.874,-49.261,-179.546,6.116,148.966
C08879=1167.963,53.123,-49.277,-179.543,6.117,148.966
C08880=1167.958,53.372,-49.293,-179.540,6.118,148.965
C08881=1167.953,53.622,-49.309,-179.538,6.119,148.965
C08882=1167.948,53.891,-49.326,-179.535,6.120,148.964
C08883=1167.942,54.159,-49.343,-179.532,6.121,148.963
C08884=1167.937,54.428,-49.360,-179.529,6.123,148.963
C08885=1167.932,54.696,-49.378,-179.527,6.123,148.962
C08886=1167.927,54.946,-49.394,-179.525,6.124,148.962
C08887=1167.922,55.196,-49.410,-179.521,6.125,148.961
C08888=1167.917,55.444,-49.426,-179.519,6.126,148.961
C08889=1167.911,55.694,-49.441,-179.516,6.127,148.960
C08890=1167.907,55.943,-49.458,-179.514,6.128,148.960
C08891=1167.902,56.193,-49.474,-179.511,6.129,148.959
C08892=1167.897,56.442,-49.490,-179.508,6.131,148.958
C08893=1167.892,56.692,-49.506,-179.506,6.131,148.958
C08894=1167.887,56.941,-49.523,-179.504,6.132,148.957
C08895=1167.882,57.191,-49.538,-179.500,6.133,148.957
C08896=1167.877,57.440,-49.555,-179.498,6.134,148.956
C08897=1167.872,57.689,-49.570,-179.495,6.135,148.956
C08898=1167.868,57.939,-49.587,-179.493,6.136,148.955
C08899=1167.862,58.188,-49.603,-179.490,6.137,148.954
C08900=1167.858,58.438,-49.619,-179.488,6.138,148.954
C08901=1167.852,58.687,-49.635,-179.485,6.139,148.953
C08902=1167.848,58.937,-49.652,-179.482,6.141,148.953
C08903=1167.842,59.186,-49.667,-179.480,6.141,148.952
C08904=1167.838,59.436,-49.684,-179.477,6.142,148.952
C08905=1167.833,59.685,-49.700,-179.474,6.143,148.951
C08906=1167.827,59.935,-49.717,-179.472,6.144,148.951
C08907=1167.822,60.184,-49.733,-179.469,6.145,148.950
C08908=1167.817,60.434,-49.749,-179.467,6.146,148.950
C08909=1167.812,60.682,-49.765,-179.464,6.147,148.949
C08910=1167.808,60.932,-49.782,-179.461,6.149,148.948
C08911=1167.803,61.181,-49.798,-179.459,6.149,148.948
C08912=1167.798,61.431,-49.814,-179.456,6.151,148.947
C08913=1167.793,61.680,-49.830,-179.453,6.151,148.947
C08914=1167.787,61.930,-49.847,-179.451,6.153,148.946
C08915=1167.782,62.179,-49.863,-179.448,6.153,148.946
C08916=1167.778,62.428,-49.880,-179.446,6.154,148.945
C08917=1167.772,62.678,-49.896,-179.443,6.156,148.945
C08918=1167.768,62.927,-49.912,-179.440,6.156,148.944
C08919=1167.764,63.177,-49.929,-179.438,6.158,148.944
C08920=1167.757,63.426,-49.945,-179.435,6.159,148.943
C08921=1167.753,63.676,-49.962,-179.432,6.160,148.943
C08922=1167.748,63.925,-49.978,-179.430,6.161,148.942
C08923=1167.743,64.174,-49.995,-179.428,6.162,148.941
C08924=1167.739,64.424,-50.011,-179.424,6.163,148.941
C08925=1167.733,64.673,-50.028,-179.422,6.164,148.940
C08926=1167.728,64.923,-50.044,-179.419,6.165,148.940
C08927=1167.723,65.172,-50.061,-179.417,6.166,148.939
C08928=1167.719,65.421,-50.077,-179.414,6.167,148.939
C08929=1167.714,65.671,-50.093,-179.411,6.168,148.938
C08930=1167.708,65.920,-50.110,-179.409,6.169,148.938
C08931=1167.704,66.170,-50.127,-179.406,6.171,148.937
C08932=1167.699,66.419,-50.143,-179.403,6.171,148.936
C08933=1167.693,66.668,-50.160,-179.401,6.173,148.936
C08934=1167.689,66.918,-50.177,-179.399,6.174,148.936
C08935=1167.683,67.167,-50.193,-179.395,6.175,148.935
C08936=1167.679,67.417,-50.209,-179.393,6.176,148.934
C08937=1167.674,67.666,-50.227,-179.390,6.177,148.934
C08938=1167.669,67.915,-50.243,-179.388,6.178,148.933
C08939=1167.664,68.165,-50.260,-179.385,6.179,148.933
C08940=1167.659,68.415,-50.277,-179.382,6.180,148.932
C08941=1167.654,68.663,-50.293,-179.380,6.181,148.932
C08942=1167.649,68.913,-50.310,-179.377,6.182,148.931
C08943=1167.644,69.163,-50.327,-179.374,6.183,148.931
C08944=1167.639,69.411,-50.343,-179.372,6.185,148.930
C08945=1167.635,69.661,-50.360,-179.370,6.185,148.930
C08946=1167.629,69.911,-50.377,-179.366,6.187,148.929
C08947=1167.624,70.159,-50.394,-179.364,6.188,148.929
C08948=1167.620,70.409,-50.410,-179.361,6.189,148.928
C08949=1167.615,70.659,-50.428,-179.359,6.190,148.927
C08950=1167.610,70.907,-50.444,-179.356,6.191,148.927
C08951=1167.604,71.157,-50.461,-179.353,6.192,148.926
C08952=1167.600,71.407,-50.478,-179.350,6.193,148.926
C08953=1167.595,71.656,-50.494,-179.348,6.194,148.925
C08954=1167.590,71.905,-50.511,-179.345,6.196,148.925
C08955=1167.585,72.155,-50.528,-179.343,6.196,148.924
C08956=1167.580,72.405,-50.545,-179.340,6.198,148.924
C08957=1167.575,72.653,-50.562,-179.337,6.199,148.923
C08958=1167.570,72.903,-50.578,-179.335,6.200,148.923
C08959=1167.565,73.153,-50.596,-179.332,6.201,148.922
C08960=1167.561,73.402,-50.612,-179.329,6.203,148.922
C08961=1167.555,73.651,-50.630,-179.327,6.203,148.921
C08962=1167.551,73.900,-50.646,-179.324,6.205,148.921
C08963=1167.545,74.150,-50.664,-179.322,6.206,148.920
C08964=1167.541,74.399,-50.680,-179.319,6.207,148.919
C08965=1167.536,74.649,-50.698,-179.316,6.208,148.919
C08966=1167.531,74.898,-50.714,-179.313,6.209,148.918
C08967=1167.525,75.148,-50.731,-179.311,6.210,148.918
C08968=1167.521,75.397,-50.749,-179.308,6.212,148.918
C08969=1167.516,75.646,-50.766,-179.306,6.212,148.917
C08970=1167.511,75.895,-50.782,-179.303,6.214,148.916
C08971=1167.506,76.145,-50.799,-179.300,6.214,148.916
C08972=1167.502,76.394,-50.817,-179.298,6.216,148.915
C08973=1167.496,76.644,-50.834,-179.295,6.217,148.915
C08974=1167.492,76.893,-50.851,-179.292,6.218,148.914
C08975=1167.486,77.142,-50.868,-179.290,6.219,148.914
C08976=1167.482,77.391,-50.885,-179.287,6.221,148.913
C08977=1167.477,77.641,-50.902,-179.285,6.221,148.913
C08978=1167.471,77.891,-50.920,-179.281,6.223,148.912
C08979=1167.467,78.140,-50.936,-179.279,6.224,148.912
C08980=1167.462,78.389,-50.954,-179.277,6.225,148.911
C08981=1167.457,78.638,-50.971,-179.274,6.226,148.911
C08982=1167.452,78.888,-50.988,-179.271,6.228,148.910
C08983=1167.447,79.137,-51.006,-179.269,6.228,148.910
C08984=1167.442,79.387,-51.022,-179.266,6.230,148.909
C08985=1167.437,79.636,-51.040,-179.264,6.231,148.909
C08986=1167.431,79.904,-51.059,-179.261,6.232,148.908
C08987=1167.427,80.173,-51.077,-179.257,6.233,148.907
C08988=1167.421,80.441,-51.096,-179.255,6.235,148.907
C08989=1167.416,80.710,-51.114,-179.252,6.236,148.906
C08990=1167.411,80.958,-51.131,-179.249,6.237,148.906
C08991=1167.406,81.208,-51.149,-179.247,6.238,148.905
C08992=1167.401,81.457,-51.167,-179.244,6.239,148.905
C08993=1167.397,81.707,-51.183,-179.242,6.240,148.904
C08994=1167.392,81.956,-51.201,-179.239,6.242,148.904
C08995=1167.386,82.206,-51.218,-179.236,6.243,148.903
C08996=1167.382,82.455,-51.235,-179.233,6.244,148.903
C08997=1167.377,82.705,-51.253,-179.230,6.246,148.902
C08998=1167.372,82.954,-51.270,-179.228,6.246,148.902
C08999=1167.367,83.204,-51.288,-179.225,6.248,148.901
C09000=1167.362,83.452,-51.305,-179.223,6.249,148.901
C09001=1167.357,83.701,-51.323,-179.220,6.250,148.900
C09002=1167.352,83.951,-51.340,-179.218,6.251,148.900
C09003=1167.347,84.200,-51.358,-179.215,6.253,148.899
C09004=1167.343,84.449,-51.375,-179.212,6.254,148.899
C09005=1167.337,84.699,-51.392,-179.210,6.255,148.898
C09006=1167.333,84.948,-51.410,-179.206,6.256,148.897
C09007=1167.327,85.198,-51.428,-179.204,6.257,148.897
C09008=1167.323,85.447,-51.445,-179.201,6.259,148.897
C09009=1167.318,85.697,-51.462,-179.199,6.259,148.896
C09010=1167.313,85.946,-51.480,-179.196,6.261,148.896
C09011=1167.308,86.195,-51.498,-179.193,6.263,148.895
C09012=1167.303,86.445,-51.516,-179.191,6.263,148.894
C09013=1167.299,86.694,-51.533,-179.188,6.265,148.894
C09014=1167.294,86.943,-51.551,-179.185,6.265,148.893
C09015=1167.289,87.193,-51.568,-179.183,6.267,148.893
C09016=1167.284,87.442,-51.586,-179.180,6.269,148.893
C09017=1167.279,87.691,-51.604,-179.177,6.269,148.892
C09018=1167.274,87.941,-51.621,-179.175,6.271,148.892
C09019=1167.269,88.190,-51.639,-179.172,6.272,148.891
C09020=1167.264,88.439,-51.657,-179.169,6.273,148.890
C09021=1167.259,88.689,-51.674,-179.167,6.274,148.890
C09022=1167.254,88.938,-51.692,-179.164,6.276,148.889
C09023=1167.249,89.187,-51.710,-179.161,6.277,148.889
C09024=1167.245,89.436,-51.728,-179.159,6.278,148.889
C09025=1167.239,89.686,-51.745,-179.156,6.279,148.888
C09026=1167.234,89.935,-51.763,-179.154,6.280,148.887
C09027=1167.229,90.184,-51.781,-179.151,6.282,148.887
C09028=1167.225,90.433,-51.799,-179.148,6.283,148.886
C09029=1167.220,90.683,-51.816,-179.146,6.284,148.886
C09030=1167.215,90.932,-51.834,-179.143,6.286,148.886
C09031=1167.210,91.181,-51.852,-179.140,6.287,148.885
C09032=1167.205,91.431,-51.870,-179.138,6.288,148.884
C09033=1167.200,91.680,-51.888,-179.135,6.290,148.884
C09034=1167.196,91.930,-51.906,-179.132,6.290,148.883
C09035=1167.191,92.179,-51.923,-179.129,6.292,148.883
C09036=1167.186,92.429,-51.941,-179.127,6.294,148.883
C09037=1167.181,92.678,-51.959,-179.124,6.294,148.882
C09038=1167.176,92.927,-51.977,-179.121,6.296,148.882
C09039=1167.171,93.176,-51.995,-179.119,6.297,148.881
C09040=1167.166,93.425,-52.013,-179.116,6.298,148.880
C09041=1167.161,93.674,-52.031,-179.113,6.300,148.880
C09042=1167.157,93.924,-52.049,-179.111,6.301,148.879
C09043=1167.152,94.173,-52.067,-179.108,6.302,148.879
C09044=1167.147,94.423,-52.086,-179.105,6.304,148.879
C09045=1167.142,94.672,-52.104,-179.103,6.305,148.878
C09046=1167.137,94.922,-52.121,-179.100,6.306,148.877
C09047=1167.132,95.171,-52.139,-179.097,6.308,148.877
C09048=1167.127,95.420,-52.157,-179.095,6.308,148.876
C09049=1167.122,95.669,-52.175,-179.092,6.310,148.876
C09050=1167.118,95.918,-52.193,-179.090,6.311,148.876
C09051=1167.113,96.168,-52.211,-179.086,6.312,148.875
C09052=1167.108,96.418,-52.230,-179.084,6.314,148.875
C09053=1167.103,96.666,-52.248,-179.082,6.315,148.874
C09054=1167.098,96.915,-52.266,-179.078,6.316,148.873
C09055=1167.093,97.165,-52.284,-179.076,6.318,148.873
C09056=1167.088,97.414,-52.302,-179.074,6.319,148.873
C09057=1167.084,97.664,-52.321,-179.070,6.320,148.872
C09058=1167.079,97.913,-52.339,-179.068,6.322,148.872
C09059=1167.074,98.162,-52.357,-179.065,6.323,148.871
C09060=1167.069,98.411,-52.375,-179.063,6.325,148.871
C09061=1167.064,98.661,-52.393,-179.060,6.326,148.870
C09062=1167.059,98.910,-52.411,-179.057,6.327,148.870
C09063=1167.054,99.160,-52.430,-179.055,6.329,148.869
C09064=1167.050,99.408,-52.448,-179.052,6.330,148.869
C09065=1167.045,99.657,-52.466,-179.049,6.331,148.868
C09066=1167.040,99.907,-52.484,-179.047,6.333,148.868
C09067=1167.035,100.157,-52.503,-179.043,6.334,148.867
C09068=1167.030,100.406,-52.521,-179.041,6.335,148.867
C09069=1167.025,100.655,-52.539,-179.039,6.336,148.866
C09070=1167.020,100.904,-52.558,-179.035,6.338,148.866
C09071=1167.016,101.154,-52.576,-179.033,6.339,148.865
C09072=1167.010,101.403,-52.595,-179.031,6.340,148.865
C09073=1167.006,101.652,-52.613,-179.027,6.342,148.864
C09074=1167.001,101.901,-52.631,-179.025,6.343,148.864
C09075=1166.997,102.151,-52.650,-179.022,6.344,148.863
C09076=1166.991,102.400,-52.668,-179.020,6.346,148.863
C09077=1166.986,102.649,-52.686,-179.017,6.347,148.862
C09078=1166.981,102.898,-52.705,-179.014,6.348,148.862
C09079=1166.977,103.148,-52.723,-179.012,6.350,148.862
C09080=1166.971,103.397,-52.742,-179.009,6.351,148.861
C09081=1166.967,103.646,-52.761,-179.006,6.352,148.860
C09082=1166.962,103.895,-52.779,-179.004,6.354,148.860
C09083=1166.957,104.145,-52.798,-179.001,6.356,148.860
C09084=1166.952,104.394,-52.816,-178.998,6.356,148.859
C09085=1166.947,104.643,-52.834,-178.996,6.358,148.859
C09086=1166.942,104.893,-52.853,-178.993,6.360,148.858
C09087=1166.938,105.142,-52.872,-178.990,6.360,148.858
C09088=1166.933,105.391,-52.890,-178.988,6.362,148.857
C09089=1166.928,105.640,-52.909,-178.985,6.364,148.857
C09090=1166.923,105.909,-52.929,-178.982,6.365,148.856
C09091=1166.917,106.177,-52.949,-178.979,6.367,148.856
C09092=1166.912,106.445,-52.969,-178.976,6.368,148.855
C09093=1166.907,106.714,-52.989,-178.973,6.370,148.855
C09094=1166.902,106.963,-53.007,-178.971,6.371,148.854
C09095=1166.898,107.212,-53.026,-178.968,6.372,148.854
C09096=1166.893,107.462,-53.045,-178.965,6.374,148.853
C09097=1166.888,107.711,-53.064,-178.963,6.375,148.853
C09098=1166.883,107.961,-53.083,-178.960,6.376,148.852
C09099=1166.878,108.209,-53.101,-178.957,6.378,148.852
C09100=1166.873,108.459,-53.119,-178.954,6.379,148.851
C09101=1166.869,108.708,-53.139,-178.952,6.380,148.851
C09102=1166.864,108.957,-53.157,-178.949,6.382,148.851
C09103=1166.858,109.206,-53.176,-178.946,6.383,148.850
C09104=1166.854,109.455,-53.195,-178.943,6.385,148.849
C09105=1166.849,109.705,-53.214,-178.941,6.386,148.849
C09106=1166.845,109.954,-53.233,-178.939,6.388,148.849
C09107=1166.839,110.204,-53.251,-178.935,6.389,148.848
C09108=1166.835,110.452,-53.270,-178.933,6.391,148.848
C09109=1166.830,110.702,-53.290,-178.931,6.392,148.847
C09110=1166.825,110.951,-53.308,-178.927,6.393,148.847
C09111=1166.820,111.201,-53.327,-178.925,6.395,148.846
C09112=1166.815,111.450,-53.345,-178.922,6.396,148.846
C09113=1166.810,111.699,-53.365,-178.920,6.397,148.845
C09114=1166.806,111.948,-53.384,-178.917,6.399,148.845
C09115=1166.800,112.197,-53.402,-178.914,6.400,148.844
C09116=1166.796,112.447,-53.421,-178.911,6.402,148.844
C09117=1166.791,112.695,-53.441,-178.909,6.403,148.844
C09118=1166.787,112.945,-53.459,-178.906,6.405,148.843
C09119=1166.781,113.194,-53.478,-178.903,6.406,148.842
C09120=1166.777,113.443,-53.497,-178.900,6.408,148.842
C09121=1166.772,113.692,-53.517,-178.898,6.409,148.842
C09122=1166.767,113.942,-53.536,-178.896,6.411,148.841
C09123=1166.762,114.191,-53.554,-178.892,6.412,148.841
C09124=1166.757,114.441,-53.574,-178.890,6.414,148.840
C09125=1166.753,114.689,-53.593,-178.887,6.415,148.840
C09126=1166.748,114.939,-53.612,-178.885,6.416,148.839
C09127=1166.742,115.188,-53.631,-178.882,6.418,148.839
C09128=1166.738,115.437,-53.650,-178.879,6.419,148.838
C09129=1166.733,115.686,-53.669,-178.876,6.421,148.838
C09130=1166.728,115.936,-53.689,-178.874,6.422,148.838
C09131=1166.724,116.184,-53.708,-178.871,6.424,148.837
C09132=1166.719,116.435,-53.727,-178.868,6.425,148.837
C09133=1166.713,116.684,-53.746,-178.865,6.427,148.836
C09134=1166.709,116.933,-53.765,-178.863,6.428,148.836
C09135=1166.704,117.182,-53.784,-178.861,6.429,148.835
C09136=1166.699,117.431,-53.804,-178.857,6.431,148.835
C09137=1166.695,117.680,-53.823,-178.855,6.432,148.834
C09138=1166.690,117.929,-53.842,-178.852,6.434,148.834
C09139=1166.685,118.178,-53.862,-178.850,6.435,148.833
C09140=1166.681,118.427,-53.881,-178.847,6.437,148.833
C09141=1166.676,118.677,-53.900,-178.844,6.438,148.832
C09142=1166.670,118.926,-53.920,-178.841,6.440,148.832
C09143=1166.666,119.175,-53.939,-178.838,6.442,148.832
C09144=1166.661,119.424,-53.958,-178.836,6.443,148.831
C09145=1166.656,119.674,-53.977,-178.834,6.444,148.831
C09146=1166.651,119.923,-53.996,-178.830,6.446,148.830
C09147=1166.646,120.172,-54.016,-178.828,6.447,148.830
C09148=1166.642,120.421,-54.036,-178.825,6.449,148.829
C09149=1166.637,120.670,-54.055,-178.822,6.451,148.829
C09150=1166.632,120.920,-54.074,-178.820,6.452,148.829
C09151=1166.627,121.169,-54.094,-178.817,6.453,148.828
C09152=1166.623,121.418,-54.113,-178.814,6.455,148.828
C09153=1166.618,121.667,-54.133,-178.812,6.456,148.827
